# B&R Automation Studio project RS15_RX_30005_r00
Automation Studio 3.0.80.31 SP01

## Configuration Config1

### Acp10map.ncm - PLC1/Motion/Acp10map.ncm
```
NcMapping (NcSwId=acp10)
  NcObject Axis3 (ModuleAddress=SL1.SS1.IF2.ST3, InterfaceType=Powerlink, Type=ncAXIS, Channel=1, InitParameter=A3_Init, AcoposParameter=A3_Par, Disabled=FALSE, ModuleDisabled=FALSE)
  NcObject SL1.SS1.IF2.ST3.VAxis1 (ModuleAddress=SL1.SS1.IF2.ST3, InterfaceType=Powerlink, Type=ncV_AXIS, Channel=1, Disabled=TRUE, ModuleDisabled=FALSE)
  NcObject Axis4 (ModuleAddress=SL1.SS1.IF2.ST3, InterfaceType=Powerlink, Type=ncAXIS, Channel=2, InitParameter=A4_Init, AcoposParameter=A4_Par, Disabled=FALSE, ModuleDisabled=FALSE)
  NcObject SL1.SS1.IF2.ST3.VAxis2 (ModuleAddress=SL1.SS1.IF2.ST3, InterfaceType=Powerlink, Type=ncV_AXIS, Channel=2, Disabled=TRUE, ModuleDisabled=FALSE)
  NcObject Axis5 (ModuleAddress=SL1.SS1.IF2.ST5, InterfaceType=Powerlink, Type=ncAXIS, Channel=1, InitParameter=A5_Init, AcoposParameter=A5_Par, Disabled=FALSE, ModuleDisabled=FALSE)
  NcObject Axis9 (ModuleAddress=SL1.SS1.IF2.ST5, InterfaceType=Powerlink, Type=ncV_AXIS, Channel=1, InitParameter=A9_Init, AcoposParameter=A9_Par, Disabled=FALSE, ModuleDisabled=FALSE)
  NcObject Axis6 (ModuleAddress=SL1.SS1.IF2.ST5, InterfaceType=Powerlink, Type=ncAXIS, Channel=2, InitParameter=A6_Init, AcoposParameter=A6_Par, Disabled=FALSE, ModuleDisabled=FALSE)
  NcObject SL1.SS1.IF2.ST5.VAxis2 (ModuleAddress=SL1.SS1.IF2.ST5, InterfaceType=Powerlink, Type=ncV_AXIS, Channel=2, Disabled=TRUE, ModuleDisabled=FALSE)
  NcObject Axis1 (ModuleAddress=SL1.SS1.IF2.ST1, InterfaceType=Powerlink, Type=ncAXIS, Channel=1, InitParameter=A1_Init, AcoposParameter=A1_Par, Disabled=FALSE, ModuleDisabled=FALSE)
  NcObject SL1.SS1.IF2.ST1.VAxis1 (ModuleAddress=SL1.SS1.IF2.ST1, InterfaceType=Powerlink, Type=ncV_AXIS, Channel=1, Disabled=FALSE, ModuleDisabled=FALSE)
  NcObject SL1.SS1.IF2.ST1.Axis2 (ModuleAddress=SL1.SS1.IF2.ST1, InterfaceType=Powerlink, Type=ncAXIS, Channel=2, Disabled=FALSE, ModuleDisabled=FALSE)
  NcObject Axis11 (ModuleAddress=SL1.SS1.IF2.ST1, InterfaceType=Powerlink, Type=ncV_AXIS, Channel=2, InitParameter=A11_Init, AcoposParameter=A11_Par, Disabled=FALSE, ModuleDisabled=FALSE)
  NcObject SL1.SS1.IF2.ST2.Axis2 (ModuleAddress=SL1.SS1.IF2.ST2, InterfaceType=Powerlink, Type=ncAXIS, Channel=2, Disabled=FALSE, ModuleDisabled=FALSE)
  NcObject SL1.SS1.IF2.ST2.VAxis2 (ModuleAddress=SL1.SS1.IF2.ST2, InterfaceType=Powerlink, Type=ncV_AXIS, Channel=2, Disabled=TRUE, ModuleDisabled=FALSE)
  NcObject Axis2 (ModuleAddress=SL1.SS1.IF2.ST2, InterfaceType=Powerlink, Type=ncAXIS, Channel=1, InitParameter=A2_Init, AcoposParameter=A2_Par, Disabled=FALSE, ModuleDisabled=FALSE)
  NcObject Axis0 (ModuleAddress=SL1.SS1.IF2.ST10, InterfaceType=Powerlink, Type=ncAXIS, Channel=1, AcoposSimulation=Off, InitParameter=A0_Init, AcoposParameter=A0_Par, Disabled=FALSE, ModuleDisabled=FALSE)
  NcObject SL1.SS1.IF2.ST10.VAxis1 (ModuleAddress=SL1.SS1.IF2.ST10, InterfaceType=Powerlink, Type=ncV_AXIS, Channel=1, Disabled=TRUE, ModuleDisabled=FALSE)
  NcObject SL1.SS1.IF2.ST10.Axis2 (ModuleAddress=SL1.SS1.IF2.ST10, InterfaceType=Powerlink, Type=ncAXIS, Channel=2, AcoposSimulation=Off, Disabled=TRUE, ModuleDisabled=FALSE)
  NcObject SL1.SS1.IF2.ST10.VAxis2 (ModuleAddress=SL1.SS1.IF2.ST10, InterfaceType=Powerlink, Type=ncV_AXIS, Channel=2, Disabled=TRUE, ModuleDisabled=FALSE)
  NcObject SL1.SS1.IF2.ST2.VAxis1 (ModuleAddress=SL1.SS1.IF2.ST2, InterfaceType=Powerlink, Type=ncV_AXIS, Channel=1, Disabled=TRUE, ModuleDisabled=FALSE)
  NcObject Axis7 (ModuleAddress=SL1.SS1.IF2.ST7, InterfaceType=Powerlink, Type=ncAXIS, Channel=1, InitParameter=A7_Init, AcoposParameter=A7_Par, Disabled=FALSE, ModuleDisabled=FALSE)
  NcObject SL1.SS1.IF2.ST7.VAxis1 (ModuleAddress=SL1.SS1.IF2.ST7, InterfaceType=Powerlink, Type=ncV_AXIS, Channel=1, Disabled=TRUE, ModuleDisabled=FALSE)
  NcObject SL1.SS1.IF2.ST7.Axis2 (ModuleAddress=SL1.SS1.IF2.ST7, InterfaceType=Powerlink, Type=ncAXIS, Channel=2, Disabled=FALSE, ModuleDisabled=FALSE)
  NcObject SL1.SS1.IF2.ST7.VAxis2 (ModuleAddress=SL1.SS1.IF2.ST7, InterfaceType=Powerlink, Type=ncV_AXIS, Channel=2, Disabled=TRUE, ModuleDisabled=FALSE)
```

## Configuration Simul_AR000

### Task classes (Cpu.sw)
```
Cyclic#1:
  A9_Basic <- BagMachine_Section.MasterAxis.A9_Init.A9_Basic.prg
  A9_Control <- BagMachine_Section.MasterAxis.A9_Init.A9_Control.prg
  A15_Basic <- BagMachine_Section.HotMicroPerf.Axis15.A15_Basic.prg
  A15_Automa <- BagMachine_Section.HotMicroPerf.Axis15.A15_Automat.prg
Cyclic#4:
  A15_Contro <- BagMachine_Section.HotMicroPerf.Axis15.A15_Control.prg
  A15_Motion <- BagMachine_Section.HotMicroPerf.Axis15.A15_MotionCycle.prg
  HMPerf_Gen <- BagMachine_Section.HotMicroPerf.HMPerf_Gen.prg
  Test_Simul <- BagMachine_Section.BagBundler.Test_Simul.prg
DataObjects: arsdmsvp, arsdmsvg, arsdmhtm, Acp10sys
NcDataObjects: A9_Par <- BagMachine_Section.MasterAxis.A9_Init.A9_Par.dob, A15_Init <- BagMachine_Section.HotMicroPerf.Axis15.A15_Init.dob, A15_Par <- BagMachine_Section.HotMicroPerf.Axis15.A15_Par.dob, A9_Init <- BagMachine_Section.MasterAxis.A9_Init.A9_Init.dob, A1_Par, A1_Init
Binaries: arsdm, webserv, Acp10map, ashwd, sysconf, arconfig, iomap, asfw, Acp10cfg, vccnum, vcnet, HMI_10, HMI_1003, vcpdvnc, vcbclass, vcgclass, vccbtn, vcpfar00, vcshared, vccline, vccdt, vcalarm, vccddbox, vcfntttf, arialbd, vctcal, vccovl, vcdsloc, visvc, vccbmp, arial, vcpdsw, vcdsint, vcfile, vccshape, HMI_1001, vcmgr, vcresman, vccstr, visapi, vcchspot, vccpopup, vcrt, HMI_1002, arialbi, vcctext, vcclbox, vccalarm
Libraries: Brsystem, NcGlobal, HGWeber, astime, runtime, powerlnk, Acp10sdc, Acp10man, Acp10par, fileio, sys_lib, asmem, standard, convert, dataobj, astcp, Acp10_MC
```

## Logical view

Binary libraries used (declarations not repeated): Acp10_MC 3.18.2, Acp10man 3.18.2, Acp10par 3.18.2, Acp10sdc 3.18.2, AsMath, AsMem, asstring, astime, Brsystem, Convert, LoopConR 2.80.0, powerlnk, sys_lib

### Global.var
```iecst
(********************************************************************
 * COPYRIGHT --
 ********************************************************************
 * File: Global.var
 * Author: pkiel
 * Created: September 02, 2009
 ********************************************************************
 * Global variables of project NewAxisControl
 ********************************************************************)
VAR
	gA : ARRAY[0..15] OF AxisBasic;
END_VAR
VAR RETAIN
	gA1_FirstHomed : BOOL;
	gA11_FirstHomed : BOOL;
END_VAR
VAR
	gA1Ref_Horn : BOOL;
	gA1Ref_PB : BOOL;
END_VAR
VAR RETAIN
	gA2_FirstHomed : BOOL;
	gA3_FirstHomed : BOOL;
END_VAR
VAR
	gA3Ref_Horn : BOOL;
	gA3Ref_PB : BOOL;
END_VAR
VAR RETAIN
	gA4_FirstHomed : BOOL;
END_VAR
VAR
	gA4Ref_PB : BOOL;
	gA4Ref_Horn : BOOL;
END_VAR
VAR RETAIN
	gA5_FirstHomed : BOOL;
END_VAR
VAR
	gA5_GearValue : REAL;
	gA5Ref_Horn : BOOL;
	gA5Ref_PB : BOOL;
END_VAR
VAR RETAIN
	gA6_FirstHomed : BOOL;
END_VAR
VAR
	gA6_GearValue : REAL;
	gA6Ref_Horn : BOOL;
	gA6Ref_PB : BOOL;
	gA8_GearValue : REAL;
	gA8Ref_Horn : BOOL;
	gA8Ref_PB : BOOL;
END_VAR
VAR RETAIN
	gA7_FirstHomed : BOOL;
END_VAR
VAR
	gA7Ref_Horn : BOOL;
	gA7Ref_PB : BOOL;
	gA13Ref_Horn : BOOL;
	gA13Ref_PB : BOOL;
	gA13_RefDone : BOOL;
	gA12Ref_Horn : BOOL;
	gA12Ref_PB : BOOL;
	gA12_RefDone : BOOL;
END_VAR
VAR RETAIN
	gA13_FirstHomed : BOOL;
	gA12_FirstHomed : BOOL;
	gA8_FirstHomed : BOOL;
	gA9_FirstHomed : BOOL;
END_VAR
VAR
	gA9Ref_Horn : BOOL;
	gA9Ref_PB : BOOL;
END_VAR
VAR RETAIN
	gA10_FirstHomed : BOOL;
END_VAR
VAR
	gA10Ref_Horn : BOOL;
	gA10Ref_PB : BOOL;
END_VAR
VAR RETAIN
	gA14_FirstHomed : BOOL;
END_VAR
VAR
	gA14_RefDone : BOOL;
END_VAR
VAR RETAIN
	gA16_FirstHomed : BOOL;
END_VAR
VAR
	gA15_RefDone : BOOL;
	gA15Ref_Horn : BOOL;
	gA15Ref_PB : BOOL;
	gA2_RefDone : BOOL;
	gA2Ref_Horn : BOOL;
	gA2Ref_PB : BOOL;
END_VAR
VAR RETAIN
	gA15_FirstHomed : BOOL;
END_VAR
VAR
	gA16_RefDone : BOOL;
	gActualMachineSpeed_BPM : REAL;
	gActualMachineSpeed_FPM : REAL;
	gAlarmReset : BOOL;
	gAlarmsOK : BOOL;
	gBagMachine_AlarmsOK : BOOL;
	gBagMachine_EstopAlarmsOK : BOOL;
	gBagMachine_GuardAlarmsOK : BOOL;
	gBagMachine_IOAlarmsOK : BOOL;
  gBagMachine_JamAlarmsOK : BOOL;
  gBagMachine_MotorAlarmsOK : BOOL;
  g_bBagMachine_GenAlarmsOK : BOOL;
	g_bBagMachine_EndReelAlarmsOK : BOOL;
	g_bBagMachine_DryerAlarmsOK : BOOL;
  g_bBagMachine_CamProfCalcOK : BOOL;
END_VAR
VAR CONSTANT
	gBlack : UINT := 0;
	gBlue : UINT := 1;
END_VAR
VAR
	gCurrentScreen : UINT;
	gDriveSupply_Ready : BOOL;
END_VAR
VAR RETAIN
	gEndPosData : ARRAY[0..15] OF MC_ENDLESS_POSITION;
END_VAR
VAR
	gEStopAlarmsOK : BOOL;
	gFastStop_OK : BOOL;
	gGeneralFaults_OK : BOOL;
  gGluerAlarmsOK : BOOL;
  g_bGenAlarmsOK : BOOL;
END_VAR
VAR CONSTANT
	gGray : UINT := 59;
	gGray1 : UINT := 250;
	gGreen : UINT := 10;
END_VAR
VAR
	gGuardAlarmsOK : BOOL;
	gGuardsOK : BOOL;
END_VAR
VAR RETAIN
	gHMI_CmdSpeed : REAL;
END_VAR
VAR
	gHMI_GoToHoldTearDrum_PB : BOOL := FALSE;
	gHMI_GoToAlarm_PB : BOOL := FALSE;
	gHMI_GoToMain_PB : BOOL := FALSE;
	gHMI_GoToMaint_PB : BOOL := FALSE;
	gHMI_GoToSetup_PB : BOOL := FALSE;
	gHMI_GoToStatus_PB : BOOL := FALSE;
	gHMI_Jog_PB : BOOL := FALSE;
	gHMI_PasswordLevel : INT;
	gHMI_Reset_PB : BOOL := FALSE;
	gHMI_Run_PB : BOOL := FALSE;
	gHMI_Stop_PB : BOOL := FALSE;
	gI_E1_Spare1 : BOOL := FALSE;
	gI_E1_Spare2 : BOOL := FALSE;
	gI_E1_Spare3 : BOOL := FALSE;
	gI_E1_Spare4 : BOOL := FALSE;
	gAI_E1_Spare1 : INT := 0;
	gAI_E1_Spare2 : INT := 0;
	gI_L3_Spare1 : BOOL := FALSE;
	gI_L3_Spare2 : BOOL := FALSE;
	gI_L3_Spare3 : BOOL := FALSE;
	gI_L3_Spare4 : BOOL := FALSE;
	gAI_L3_Spare1 : INT := 0;
	gAI_L3_Spare2 : INT := 0;
	gI_230Vac_OK : BOOL := FALSE;
	gI_AirPressureOK : BOOL := FALSE;
	gI_EstopPB_1 : BOOL := FALSE; (*+R4*)
	gI_EstopPB_2 : BOOL := FALSE; (*+R3*)
	gI_EstopPB_3 : BOOL := FALSE; (*+R1*)
	gI_EstopPB_4 : BOOL := FALSE; (*+R2*)
	gI_EstopPB_5 : BOOL := FALSE; (*+R1A*)
	gI_EstopPB_Unwind : BOOL := FALSE;
	gI_FasterPB_1 : BOOL := FALSE;
	gI_FstopPB_1 : BOOL := FALSE;
	gI_GSW_Door1 : BOOL := FALSE;
	gI_GSW_Door2 : BOOL := FALSE;
	gI_GSW_Drum : BOOL := FALSE;
	gI_GSW_PerfDoors : BOOL := FALSE;
	gI_GSW_PerfDoor2 : BOOL := FALSE;
	gI_GSW_RSEntry : BOOL := FALSE;
	gI_GSW_SlittingDoor : BOOL := FALSE;
	gI_GSW_Tearing : BOOL := FALSE;
	gI_JamPE_RS : BOOL := FALSE;
	gI_JogPB_1 : BOOL := FALSE;
	gI_MP_DrumFan : BOOL := FALSE;
	gI_MP_GlueSlowRotation : BOOL := FALSE;
	gI_MP_PerfFan : BOOL := FALSE;
	gI_MP_Vacuum : BOOL := FALSE;
	gI_PB_MachineStart : BOOL := FALSE;
	gI_ResetPB_1 : BOOL := FALSE;
	gCmd_ResetPBGen : BOOL := FALSE; (*General reset all failures*)
	gI_SafetyRelay_EStopOK : BOOL := FALSE;
	gI_SafetyRelay_GuardOK : BOOL := FALSE;
	gI_SlowerPB_1 : BOOL := FALSE;
	gI_SlowerPB_2 : BOOL := FALSE;
	gI_SS_DrumNeg : BOOL := FALSE;
	gI_SS_DrumPos : BOOL := FALSE;
	gI_SS_ExitTableFaster : BOOL := FALSE;
	gI_SS_ExitTableSlower : BOOL := FALSE;
	gI_SS_GluePanUpDown : BOOL := FALSE;
	gI_SS_HoldingNeg : BOOL := FALSE;
	gI_SS_HoldingPos : BOOL := FALSE;
	gI_SS_MainPowerOff : BOOL;
	gI_SS_MainPowerOn : BOOL := FALSE;
	gI_SS_PerfNeg : BOOL := FALSE;
	gI_SS_PerfPos : BOOL := FALSE;
	gI_SS_SeamGlueOnOff : BOOL := FALSE;
	gI_PrintOn_PB : BOOL := FALSE;
	gI_PrintOff_PB : BOOL := FALSE;
	gI_SS_TearingNeg : BOOL := FALSE;
	gI_SS_TearingPos : BOOL := FALSE;
	gI_SS_WebEntryNipOff_1 : BOOL := FALSE;
	gI_SS_WebEntryNipOff_2 : BOOL := FALSE;
	gI_SS_WebEntryNipOn_1 : BOOL := FALSE;
	gI_SS_WebEntryNipOn_2 : BOOL := FALSE;
	gI_SS_WebExitNip : BOOL := FALSE;
	gI_StopPB_1 : BOOL := FALSE;
	gI_StopPB_2 : BOOL := FALSE;
	gI_StopPB_3 : BOOL := FALSE; (*Stop PB on +R2 panel*)
	gI_JogPB_2 : BOOL := FALSE; (*Footswitch Job*)
	gI_JogPB_3 : BOOL := FALSE; (*Flexo press Job*)
	gI_WebBreakPE_1 : BOOL := FALSE;
	gI_WebBreakPE_2 : BOOL := FALSE;
	gI_EstopPB_FlexoPress : BOOL := FALSE;
	gI_UNW_EndReelPolyPE : BOOL := FALSE;
	gI_UNW_EndReelPapPE : BOOL := FALSE;
	gI_SS_UNW_ForkUp : BOOL := FALSE;
	gI_SS_UNW_ForkDown : BOOL := FALSE;
	gI_SS_UNW_Brake : BOOL := FALSE;
	gI_MP_UNW_HydroPump : BOOL := FALSE;
	gI_SS_UNW_HotGlue : BOOL := FALSE;
	gI_SS_FP_NipRol : BOOL := FALSE;
	gI_MP_FP_MotorFan : BOOL := FALSE;
	gI_FP_PrintOn_PB : BOOL := FALSE;
	gI_FP_PrintOff_PB : BOOL := FALSE;
	gI_MP_FP_SlowRot5 : BOOL := FALSE;
	gI_MP_FP_SlowRot6 : BOOL := FALSE;
	gI_GSW_FP_Doors : BOOL := FALSE;
	gI_GSW_FP_Gates : BOOL := FALSE;
	gI_MP_FP_SlowRot1 : BOOL := FALSE;
	gI_MP_FP_SlowRot3 : BOOL := FALSE;
	gI_MP_FP_SlowRot2 : BOOL := FALSE;
	gI_MP_FP_SlowRot4 : BOOL := FALSE;
	gI_HMP_BrushReturnPE : BOOL := FALSE;
	gI_HMP_ProtecDownPE : BOOL := FALSE;
	gI_SS_HMPerfNeg : BOOL := FALSE;
	gI_SS_HMPerfPos : BOOL := FALSE;
	gI_HMP_On_PB : BOOL := FALSE;
	gI_HMP_Off_PB : BOOL := FALSE;
	gI_HMP_EStopPB : BOOL := FALSE;
	gI_SS_HMP_Heating : BOOL := FALSE;
	gI_GSW_HMPerf : BOOL := FALSE;
	gI_SS_HMP_ManuProtecDown : BOOL := FALSE;
	gI_HMP_ManuBrushForward_PB : BOOL := FALSE;
	gI_HMP_WebBreakPE : BOOL := FALSE;
	gI_HMP_JogPB : BOOL := FALSE;
	gI_L15_Spare1 : BOOL := FALSE;
	gI_L15_Spare2 : BOOL := FALSE;
	gI_L15_Spare3 : BOOL := FALSE;
	gI_L15_Spare4 : BOOL := FALSE;
	gI_SS_3W_GlueOn : BOOL := FALSE;
	gI_SS_3W_Glue2 : BOOL := FALSE;
	gI_MP_HP_WasteSuction : BOOL := FALSE;
	gI_3W_EndReelPolyPE : BOOL := FALSE;
	gI_MP_3W_Fan : BOOL := FALSE;
	gI_3W_EStopPB : BOOL := FALSE;
	gI_GSW_3W : BOOL := FALSE;
	gI_SS_3W_FanOnOff : BOOL := FALSE;
	gI_DRY_Thermostat : BOOL := FALSE;
	gI_MP_DRY_Blower : BOOL := FALSE;
	gI_MP_DRY_Heater : BOOL := FALSE;
	gI_E1_Spare6  : BOOL := FALSE;
  gI_E1_Spare5  : BOOL := FALSE;
  gI_E1_Spare7  : BOOL := FALSE;
  gI_E1_Spare8  : BOOL := FALSE;
  gI_E1_Spare9  : BOOL := FALSE;
  gI_E1_Spare10 : BOOL := FALSE;
	gI_L3_Spare5 : BOOL := FALSE;
	gI_L3_Spare6 : BOOL := FALSE;
	gI_L3_Spare7 : BOOL := FALSE;
	gI_GSW_CMPerfDoor : BOOL := FALSE;
	gI_GSW_CMPerfGates : BOOL := FALSE;
	gI_MP_EB_WasteSuction : BOOL := FALSE;
	gI_SS_EnvBagNeg : BOOL := FALSE;
	gI_SS_EnvBagPos : BOOL := FALSE;
	gI_SS_TearEBNeg : BOOL := FALSE;
	gI_SS_TearEBPos : BOOL := FALSE;
	gAI_DRY_Pt100_Temp : INT;
END_VAR
VAR RETAIN
	gMachineTime : HourMeter;
END_VAR
VAR
	gMaintDropdown : UINT;
	gMaintScreenChange : BOOL;
	gManualMode_On : BOOL;
	gMotorAlarmsOK : BOOL;
	gNever : BOOL;
	gNever1 : BOOL; (*D.M. 05/08/2011 Inibit function BrownPaper_14542*)
END_VAR
VAR RETAIN
	gPassword : PasswordLevel;
END_VAR
VAR
	gPerf_On : BOOL;
	gPerf_ParkRequest : BOOL;
END_VAR
VAR RETAIN
	gPerf_ParkRequired : BOOL;
END_VAR
VAR
	gPerfSelect_Large : BOOL;
	gPowerUp_Complete : BOOL;
END_VAR
VAR CONSTANT
	gPurple : UINT := 62;
END_VAR
VAR
	gQ_E1_Spare1 : BOOL := FALSE;
	gQ_E1_Spare2 : BOOL := FALSE;
  gQ_E1_Spare3 : BOOL := FALSE;
  gQ_E1_Spare4 : BOOL := FALSE;
  gQ_E1_Spare5 : BOOL := FALSE;
  gQ_E1_Spare6 : BOOL := FALSE;
	gAQ_E1_Spare1 : INT := 0;
	gAQ_E1_Spare2 : INT := 0;
	gQ_L3_Spare1 : BOOL := FALSE;
	gQ_L3_Spare2 : BOOL := FALSE;
  gQ_L3_Spare3 : BOOL := FALSE;
  gQ_L3_Spare4 : BOOL := FALSE;
  gQ_L3_Spare5 : BOOL := FALSE;
  gQ_L3_Spare6 : BOOL := FALSE;
	gAQ_L3_Spare1 : INT := 0;
	gAQ_L3_Spare2 : INT := 0;
	gQ_CMD_ColdGluePressure : INT := 0;
	gQ_CMD_EjectionTableMotor : INT := 0;
	gQ_CMD_HotGluePressure : INT := 0;
	gQ_CMD_RS_GluePressure : INT := 0;
	gQ_CMD_UNW_GluePressure : INT := 0;
	gQ_CMD_3W_GluePressure : INT := 0;
	gQ_CMD_OtherRS_GluePressure : INT := 0;
	gQ_CMD_RS_ExitTableSpeed : INT := 0;
	gQ_CON_GlueSlowRotation : BOOL := FALSE;
	gQ_CON_Vacuum : BOOL := FALSE;
	gQ_CR_ColdGlue : BOOL := FALSE;
	gQ_CR_ColdGlueSelect : BOOL := FALSE;
	gQ_CR_EstopReset : BOOL := FALSE;
	gQ_CR_GuardBypass : BOOL := FALSE;
	gQ_CR_HotGlue : BOOL := FALSE;
	gQ_CR_HotGlueSelect : BOOL := FALSE;
	gQ_CR_MainPowerOn : BOOL := FALSE;
	gQ_CR_UnwinRegEnable : BOOL := FALSE; (*Enable regulation on the unwinder*)
	gQ_CR_WarningHorn : BOOL := FALSE;
	gQ_CR_WatchDog : BOOL := FALSE;
	gQ_PL_GenFailure : BOOL := FALSE;
	gQ_PL_MainPower : BOOL := FALSE;
	gQ_SOL_BagCount : BOOL := FALSE;
	gQ_SOL_GluePan : BOOL := FALSE;
	gQ_SOL_WebEntryNip : BOOL := FALSE;
	gQ_SOL_WebExitNip : BOOL := FALSE;
	gQ_CR_UNW_HydroPump : BOOL := FALSE;
	gQ_CR_HotColdRSGlueSelect : BOOL := FALSE;
	gQ_CR_HotColdOtherRSGlueSelect : BOOL := FALSE;
	gQ_CR_UNW_Brake : BOOL := FALSE; (*MEROBEL device input B*)
	gQ_CR_FP_NipRol : BOOL := FALSE;
	gQ_CR_FP_Print : BOOL := FALSE;
	gQ_CR_UNW_PIDRegul : BOOL := FALSE; (*MEROBEL device input A*)
	gQ_CR_UNW_ForkUp : BOOL := FALSE;
	gQ_CR_UNW_ForkDown : BOOL := FALSE;
	gQ_CR_RS_Glue : BOOL := FALSE;
	gQ_CR_UNW_Glue : BOOL := FALSE;
	gQ_SOL_HMP_BrushForward : BOOL := FALSE;
	gQ_SOL_HMP_ProtecDown : BOOL := FALSE;
	gQ_HMP_LightOn : BOOL := FALSE;
	gQ_HMP_Heater : BOOL := FALSE;
	gQ_CR_3W_GlueOn : BOOL := FALSE;
	gQ_CR_3W_Glue2 : BOOL := FALSE;
	gQ_CR_3W_Fan : BOOL := FALSE;
	gQ_CR_HP_WasteSuction : BOOL := FALSE;
	gQ_CR_DRY_Blower : BOOL := FALSE;
	gQ_CR_DRY_HeatRegul : BOOL := FALSE;
	gQ_CR_DRY_HeatContinu : BOOL := FALSE;
	gQ_CR_EB_WasteSuction : BOOL := FALSE;
	gQ_CR_UNW_Lock : BOOL := FALSE;
END_VAR
VAR RETAIN
	gRecipeActive : Recipe := (rEnvB_PerfSize_in:=18.897); (*Default Envelope Bag Perf Size = 480mm Customer Pyrollpack_14661*)
	gRecipeBase : ARRAY[0..50] OF Recipe;
END_VAR
VAR
	gRecipeChange : BOOL;
	gRecipeCntl : RECIPE_CNTL_typ;
END_VAR
VAR CONSTANT
	gRed : UINT := 51;
END_VAR
VAR RETAIN
	gReg : ARRAY[0..15] OF Registration;
END_VAR
VAR
	gInchMetric_Ind : UINT; (*=1:Inch, =2:Metric*)
	gIOAlarmsOK : BOOL;
	gJamAlarmsOK : BOOL;
	gWebBreakAlarmsOK : BOOL;
	gJog_Horn : BOOL;
	gJog_ToZeroFiltered : BOOL;
	gRun_Stop : BOOL;
	gJog_Stop : BOOL;
	gJog_ToZeroSpeed : BOOL;
	gMachine_Jog : BOOL;
	gMachine_Run : BOOL;
	gMachineMaxSpeedLimit : REAL;
	gMachineMinSpeedLimit : REAL;
	gRepeatChange : BOOL;
	gRun_Horn : BOOL;
	gRun_ToZeroSpeed : BOOL;
	gScreenControl : UINT;
	gServoAxesOK : BOOL;
	gSetupMode_On : BOOL;
	gSetupPermissive : BOOL;
END_VAR
VAR RETAIN
	gSP_A : ARRAY[0..15] OF AxisSP := [(HomeOffset:=0.0,PhaseOffset:=0.0,Diameter:=0.0,ParkPosition:=0.0,MatchedSpeed:=0.0,AbsoluteOffset:=0.0,rZoneBefPerf_in:=0.0,rZoneAftPerf_in:=0.0),(HomeOffset:=120.0,ParkPosition:=120.0,MatchedSpeed:=60.0),(HomeOffset:=0.0,PhaseOffset:=0.0,Diameter:=0.0,ParkPosition:=0.0,MatchedSpeed:=0.0,AbsoluteOffset:=0.0,rZoneBefPerf_in:=0.0,rZoneAftPerf_in:=0.0),2((HomeOffset:=20.0)),2((HomeOffset:=0.0,PhaseOffset:=0.0,Diameter:=0.0,ParkPosition:=0.0,MatchedSpeed:=0.0,AbsoluteOffset:=0.0,rZoneBefPerf_in:=0.0,rZoneAftPerf_in:=0.0)),(HomeOffset:=20.0),(HomeOffset:=20.0,PhaseOffset:=0.0,Diameter:=0.0,ParkPosition:=0.0,MatchedSpeed:=0.0,AbsoluteOffset:=0.0,rZoneBefPerf_in:=0.0,rZoneAftPerf_in:=0.0),4((HomeOffset:=0.0,PhaseOffset:=0.0,Diameter:=0.0,ParkPosition:=0.0,MatchedSpeed:=0.0,AbsoluteOffset:=0.0,rZoneBefPerf_in:=0.0,rZoneAftPerf_in:=0.0)),(HomeOffset:=20.0,PhaseOffset:=0.0,Diameter:=0.0,ParkPosition:=0.0,MatchedSpeed:=0.0,AbsoluteOffset:=0.0,rZoneBefPerf_in:=0.0,rZoneAftPerf_in:=0.0),2((HomeOffset:=0.0,PhaseOffset:=0.0,Diameter:=0.0,ParkPosition:=0.0,MatchedSpeed:=0.0,AbsoluteOffset:=0.0,rZoneBefPerf_in:=0.0,rZoneAftPerf_in:=0.0))];
	gSP_EnvBPerf : AxisSP; (*Envelope Bag Perf*)
	gSP_StandPerf : AxisSP; (*Standard Perf*)
	gSP_CmdSpeed : REAL;
	gSP_ColdGlue : Glue;
	gSP_RSGlue : Glue;
	gSP_OtherRSGlue : Glue;
	gSP_GlueTrayAutoSpeed : REAL;
	gSP_HotGlue : Glue;
	gSP_PerfCylSelect : BOOL; (*Perf Size selection =0:Small; =1:Large*)
	gSP_PerfKnifeCount : REAL;
	gSP_TubeSelect : BOOL;
END_VAR
VAR
	gStopPosition : REAL;
	gStopStringOK : BOOL;
	gTubeSelect_2 : BOOL;
	gUnwindLowRoll_Stop : BOOL;
	gBagMachine_WebBreakOK : BOOL;
	gWebBreakBypass_On : BOOL;
	g_bEndReelPapBypass_On : BOOL;
	g_bEndReelPolyBypass_On : BOOL;
	g_rActualSizePerf_in : REAL; (*Actual perimeter of the Perf, in inch*)
	g_bPerfInMatchedSpeed : BOOL;
	g_bMainPower_On : BOOL;
	g_bMainPower_OnDelay : BOOL;
  g_bCamPerfCalc_Error : BOOL;
  g_bCamPerfCalcReset : BOOL;
  g_uiCalcCamPerfErrorID : UINT;
  g_bMachineRun : BOOL;
  g_bCameProf_OK : BOOL;
  g_uiIndexCamProfPerf : UINT;
  g_uiGetPosCamProfErrorID_1 : UINT;
  g_uiGetPosCamProfErrorID_2 : UINT;
  g_uiGetPosCamProfErrorID_3 : UINT;
  g_uiHomCamProfErrorID : UINT;
  g_bGetMaPosCamProfError_1 : BOOL;
  g_bGetMaPosCamProfError_2 : BOOL;
  g_bHomeCamProfError : BOOL;
  g_uiGetPosCamProfErrorID : UINT;
  g_bGetMaPosCamProfError : BOOL;
  g_bGetSlPosCamProfError : BOOL;
  g_rPosParkMasterCam : REAL ;
	g_bIndSynchroHTD_OK : BOOL; (*Indicator synchro Holding, Tearing and Drum axis is completed*)
	g_iMachType : INT; (*Machine type : =1:RS26, =2:RS15, =3:RS25*)
	g_iFlexoType : INT; (*Flexo type : =0:Metric, =1:8DP, =2:10DP, =3:1/4"*)
	g_bIndEStop : BOOL; (*EStop active*)
	g_bIndEStopStandstill : BOOL; (*EStop when machine at standstill*)
	g_bIndStopFault : BOOL; (*Machine stopping on fault condition*)
  g_bUnwindInMach : BOOL;
  g_bUnwindEndRelPapInMach : BOOL;
  g_bUnwindEndRelPolyInMach : BOOL;
	g_bFP_IndSpeedLimit : BOOL; (*Speed limited because max speed Flexo Press reached*)
	g_rNumbPliers : REAL; (*Number of pliers on the Drum, 4 or 2*)
	g_bNumPliersChange : BOOL;
	g_bNumPliersChange2to4 : ARRAY[1..3] OF BOOL; (*Change number of pliers on the Drum, from 2 to 4*)
	g_bNumPliersChange4to2 : ARRAY[1..3] OF BOOL; (*Change number of pliers on the Drum, from 4 to 2*)
	g_bChangeModTearingReq : BOOL; (*Change modulus on tearing axis request*)
	g_bChangeModTearEBReq : BOOL; (*Change modulus on Tearing Envelope Bag axis request*)
	g_bChangeModDrumReq : BOOL; (*Change modulus on tearing axis request*)
	g_bRedefPosdTearingReq : BOOL; (*Redefinition of the position on Tearing axis request*)
	g_bRedefPosDrumReq : BOOL; (*Redefinition of the position on Drum axis request*)
	g_bSynchroAxisOK : BOOL; (*All axis are synchro*)
	g_bSynchroAxisInProgress : BOOL; (*Synchro axis in progress*)
	g_rMaxBagSize_Inch : REAL;
	g_rMinBagSize_Inch : REAL;
	g_bSplashDone : BOOL;
	g_b3WebUnitInMach : BOOL;
	g_bFP_NipRolAutoOff : BOOL;
	g_bFP_GuardFault : BOOL;
	g_bLockSP_OffsetPrintRol : BOOL;
	g_bFP_SP_Offset : BOOL; (*Change Offset of the Flexo with set point motion*)
	g_rPrintRolCalcPos_deg : REAL; (*Calculated position of the printing rolle, in °*)
	g_rPrintRolCalcPos_in : REAL; (*Calculated position of the printing rolle, in inch*)
	g_HMI_Cmd_ManuTimSetPlus : BOOL;
	g_bCondManuTimSet : BOOL;
	g_bStartOffsetAuto : BOOL;
	g_rZGearRepFP : REAL := 40.0; (*Current tooth number of the gear on the Flexo Press*)
	g_bCmdShiftA : ARRAY[1..15] OF BOOL; (*Command shift Axe[n]*)
	g_iCountPerfShift : ARRAY[1..2] OF INT; (*Counter of Perf shifting in order to match with printing position*)
	g_iNumBagPerfTear : INT; (*Num bags between Perf en teraing > gr_rDistPerfTear_mm / BagSize example : 3800/200 = 19*)
	g_iArrayBagPerfTear : ARRAY[0..C_iMaxBagPerfTear] OF INT; (*Array of bags between Perf and tearing, +1 for positive shift and -1 for negative shift*)
	g_iArrayBagPerfTearNul : ARRAY[0..C_iMaxBagPerfTear] OF INT := [C_iMaxBagPerfTear(0)]; (*Array with all elements C_iMaxBagPerfTear =0*)
	gr_rIndEnvB2AxTear1 : BOOL := 0; (*Envelope Bag 2 Axes, indicator tearin on the first station (tube lenght > gr_rEnvBSizeTear2_1_mm), =0:NO; =1:YES *)
	g_bPerfShiftPos : BOOL;
	g_iPerfShiftPos : INT;
	g_bCycManTimeSetOn : BOOL; (*Indicator at least one manual timing setting is active*)
	g_bIndPhasDrumInact : BOOL := 0; (*Indicator phasing Drum inactive*)
	g_rZGearCMPerf : REAL; (*Current number of tooth on the gear which drive the Cold Micro Perf Tool*)
	g_rSizeCMPerf : REAL; (*Current number of tooth on the gear which drive the Cold Micro Perf Tool*)
	g_rSizeCMPerfRol_mm : REAL; (*Perimeter of the shaft which drive the Cold Micro Perf Tool, in mm*)
	g_iCMPerfType : INT; (*Cold Micro Perf type : =0:Metric, =1:8DP, =2:10DP, =3:1/4"*)
	g_stHMPerfCyc : CycHMPerf;
	g_bHMP_WebBreakBypass_On : BOOL;
	g_bHMP_CamOK : BOOL;
	g_bHMP_CamCalcReset : BOOL;
	g_bHMP_CamErrorGen : BOOL;
	g_bHMP_CamCalc_Error : BOOL;
	g_uiHMP_CalcCamErrorID : UINT;
	g_bHMP_CamDownl_Error : BOOL;
	g_uiHMP_DownlCamErrorID : UINT;
	g_bHMP_CmdPhasing : BOOL; (*Hot Micro Perf Phasing command to set the Offset when synchronizing*)
	g_bHMP_PhasInProgres : BOOL; (*Hot Micro Perf Phasing in progress to set the Offset when synchronizing*)
	g_rHMP_SP_Phasing : REAL; (*Hot Micro Perf Phasing Phasing Set Point to set the Offset when synchronizing, in Deg*)
	g_bDryerInMach : BOOL;
	g_bHeatDryInMach : BOOL;
	g_bSelDryerProd : BOOL;
	g_usiAI_DRY_Pt100_TempStatus : USINT;
	g_DRY_bTempSensorAlarm : BOOL;
	g_DRY_bHeaterAlarm : BOOL;
  g_DRY_bBlowerAlarm : BOOL;
  g_DRY_bActHeat : BOOL;
  g_DRY_bIndCooling : BOOL;
  g_DRY_bMemPowerOff : BOOL;
  g_DRY_bFlash : BOOL ;
	g_iPerfType : INT;
	g_bEnvBagSelectChang : BOOL;
	g_EnvB_bWasteSucMPAlarm : BOOL;
	g_EnvB_iHoldTearEnvBCase : INT;
END_VAR
VAR CONSTANT
	C_iRS26 : INT := 1;
	C_iRS15 : INT := 2;
	C_iRS25 : INT := 3;
	C_iM : INT := 0;
	C_i8DP : INT := 1;
	C_i10DP : INT := 2;
	C_i1_4P : INT := 3;
	gWhite : UINT := 15;
	gViolet_5 : UINT := 5;
	gYellow : UINT := 46;
	C_rMaxAna : REAL := 32767.0;
	C_iMaxBagPerfTear : INT := 39; (*Num max bags between > MaxDistPerfTear / MinBagSize = Around(4000/105) = 39*)
END_VAR
VAR RETAIN
	g_rBagSize1to2SPerf_in : REAL := 7.480; (*Bag Size for switching 1 --> 2 blades on the Perfo (1if >; 2 if <=) case Small Perfo, in in*)
	g_rBagSize1to2LPerf_in : REAL := 10.236; (*Bag Size for switching 1 --> 2 blades on the Perfo (1if >; 2 if <=) case Large Perfo, in mm*)
	g_rLinSpeedMin_ftmin : REAL := 32.808; (*Value of the Minimum Speed, in ft/min*)
END_VAR
VAR CONSTANT
	PI : REAL := 3.14159;
END_VAR
VAR
	g_rLinSpeedMin_bgmin        : REAL := 0.0; (*Value of the Minimum Speed, in bg/min*)
	g_rBagSize1to2SPerf_mm      : REAL := 190.0; (*Bag Size for switching 1 --> 2 blades on the Perfo (1if >; 2 if <=) case Small Perfo, in mm*)
	g_rBagSize1to2LPerf_mm      : REAL := 260.0; (*Bag Size for switching 1 --> 2 blades on the Perfo (1if >; 2 if <=) case Large Perfo, in mm*)
	g_rLinSpeedMin_mmin         : REAL := 10.0; (*Value of the Minimum Line Speed, in m/min*)
	g_rMaxSpeedMin_bpm          : REAL := 35.0; (*Value of the max bag/min at minimum speed, in bag/min*)
	g_rMaxSpeedSynchro_bpm      : REAL := 8.0; (*Value of the max bag/min when synchronising, in bag/min*)
	g_rMaxJogDecel_bpmm         : REAL := 1200.0; (*Value of the max Jog deceleration, in bag/min²*)
	g_rLinSpeedSP_AccRS26           : REAL := 600.0; (*Value of Line Speed SP accel, in m/min²*)
	g_rLinSpeedSP_DecRS26           : REAL := 600.0; (*Value of Line Speed SP decel, in m/min²*)
	g_rLinSpeedSP_JogDecRS26        : REAL := 2500.0; (*Value of Line Speed SP Jog decel, in m/min²*)
	g_rLinSpeedSP_EStopDecRS26      : REAL := 6000.0; (*Value of Line Speed SP EStop decel, in m/min²*)
	g_rLinSpeedSP_GuardFaultDecRS26 : REAL := 4500.0; (*Value of Line Speed SP Guard Fault decel, in m/min²*)
	g_rLinSpeedSP_WebBreakDecRS26   : REAL := 5200.0; (*Value of Line Speed SP EStop decel, in m/min²*)
	g_rLinSpeedSP_GenFaultDecRS26   : REAL := 3000.0; (*Value of Line Speed SP General Fault decel, in m/min²*)
  g_rLinSpeedSP_FStopDecRS26      : REAL := 1800.0; (*Value of Line Speed SP Fast Stop decel, in m/min²*)
  g_rLinSpeedSP_AccRS15           : REAL := 33.3; (*Value of Speed SP accel, in m/min/s => 0-->1000bag/min in 30s*)
  g_rLinSpeedSP_DecRS15           : REAL := 33.3; (*Value of Speed SP decel, in m/min/s => 0-->1000bag/min in 30s*)
  g_rLinSpeedSP_JogDecRS15        : REAL := 140.0; (*Value of SP Jog decel, in m/min/s => 1000-->0bag/min in 7s*)
  g_rLinSpeedSP_EStopDecRS15      : REAL := 333; (*Value of Speed SP EStop decel, in m/min/s => 1000-->0bag/min in 3s*)
  g_rLinSpeedSP_GuardFaultDecRS15 : REAL := 250.0; (*Value of Speed SP Guard Fault decel, in m/min/s => 1000-->0bag/min in 4s*)
  g_rLinSpeedSP_WebBreakDecRS15   : REAL := 250.0; (*Value of Speed SP EStop decel, in m/min/s => 1000-->0bag/min in 4s*)
  g_rLinSpeedSP_GenFaultDecRS15   : REAL := 167.0; (*Value of Speed SP General Fault decel, in m/min/s => 1000-->0bag/min in 6s*)
  g_rLinSpeedSP_FStopDecRS15      : REAL := 100.0; (*Value of Speed SP Fast Stop decel, in m/min/s => 1000-->0bag/min in 10s*)
  g_rSizeEntryPullRol_mm      : REAL := 400.0; (*Perimeter of the entry pull roll, in mm*)
	g_rSizeExitPullRol_mm       : REAL := 320.0; (*Perimeter of the exit pull roll, in mm*)
	g_rSizeLPerf_mm       : REAL := 400.0; (*Perimeter of the large Perf, in mm*)
	g_rSizeSPerf_mm       : REAL := 270.0; (*Perimeter of the small Perf, in mm*)
	g_rSizeDrum_mm        : REAL := 1680.0; (*Perimeter of the Drum, in mm*)
	g_rZGearRepFP_M       : REAL := 40.0; (*Tooth number of the gear on the Flexo Press in case Metric*)
	g_rZGearRepFP_8DP     : REAL := 40.0; (*Tooth number of the gear on the Flexo Press in case 8DP*)
	g_rZGearRepFP_10DP    : REAL := 50.0; (*Tooth number of the gear on the Flexo Press in case 10DP*)
	g_rZGearRepFP_1_4P    : REAL := 65.0; (*Tooth number of the gear on the Flexo Press in case 1/4"*)
	g_rZGearCMPerf_M      : REAL := 50.0; (*Tooth number of the gear on the shaft which drive the Cold Micro Perf Tool in case Metric*)
	g_rZGearCMPerf_8DP    : REAL := 50.0; (*Tooth number of the gear on the shaft which drive the Cold Micro Perf Tool in case 8DP*)
	g_rZGearCMPerf_10DP   : REAL := 63.0; (*Tooth number of the gear on the shaft which drive the Cold Micro Perf Tool in case 10DP*)
	g_rZGearCMPerf_1_4P   : REAL := 81.0; (*Tooth number of the gear on the shaft which drive the Cold Micro Perf Tool in case 1/4"*)
  g_rMaxBagSize_RS15_mm : REAL := 400.0;
  g_rMinBagSize_RS15_mm : REAL := 105.0;
  g_rMaxBagSize_RS26_mm : REAL := 760.0;
  g_rMinBagSize_RS26_mm : REAL := 160.0;
  g_rMaxBagSize_EnvB_mm : REAL := 760.0;
  g_rMinBagSize_EnvB_mm : REAL := 240.0;
END_VAR

VAR RETAIN
  g_rSizeEnvBPerf_mm : REAL := 520.0; (*Perimeter of the Envelope Bag Perf, in mm*)
END_VAR

VAR RETAIN
	gr_rMachMaxSpeed_BPM        : REAL := 1000.0; (*Parameter : machine max speed, in Bag/min*)
	gr_rHoldAxContactZone       : REAL := 22.0;   (*Parameter : zone where Holding Axis is in contact, in Deg*)
	gr_rTearAxContactZone       : REAL := 52.0;   (*Parameter : zone where Tearing Axis is in contact with the Bag, in Deg*)
	gr_rDrumAxContactZone       : REAL := 50.0;   (*Parameter : zone where Drum Axis is in contact with the blade, in Deg*)
	gr_rEnvBAxContactZone       : REAL := 26.0;   (*Parameter : zone where Envelope Bag Axis is in contact with the Bag, in Deg*)
	gr_rTearEBAxContactZone     : REAL := 52.0;   (*Parameter : zone where Tearing of the Envelope Bag Axis is in contact with the Bag, in Deg*)
	gr_rPosHoldBag              : REAL := 11.0;   (*Position of the Holding axis when the shaft is vertical, the bag is maintained, in°*)
	gr_rPosTearBag              : REAL := 26.0;   (*Position of the Tearing axis when the shaft is vertical, the bag is Teared, in°*)
	gr_rPosGripBag              : REAL := 25.0;   (*Position of the Drum axis when the blade is in the gripper, the bag is gripped, in°*)
	gr_rPosEnvBHoldBag          : REAL := 355.0;  (*Position of the Envelope Bag axis when the shaft is vertical, the bag is maintained and the nidles are outside, in°*)
	gr_rPosTearEBTearBag        : REAL := 18.0;   (*Position of the Tearing Envelope Bag axis when the shaft is vertical, the bag is Teared, in°*)
	gr_rAxisTimSet_SP_Vel       : REAL := 12;     (*Set point Velocity for Axis manual timing setting cycle, in Axis round/min*)
	gr_rAxisTimSet_SP_Acc       : REAL := 1200;   (*Set point Acceleration for Axis manual timing setting cycle, in Axis round/min²*)
	gr_rAxisTimSet_SP_Dec       : REAL := 3000;   (*Set point Deceleration for Axis manual timing setting cycle, in Axis round/min²*)
	gr_rMaxRangeWebDraw         : REAL := 1;      (*Max range for web draw modification on pull roll, in %*)
	gr_rLimOffsetRunVal         : REAL := 0.1;    (*Limit the max value of Offset changing when Running, in % of the Repeat*)
	gr_rIncrOffsetAxeRun        : REAL := 1.0;    (*Increment offset axis changing when Running, in mm/bag*)
	gr_tJogHornDur              : TIME := T#1s;   (*Horn duration in Jog, in s*)
	gr_tRunHornDur              : TIME := T#1s500ms; (*Horn duration in Run, in s*)
  gr_rMaxLSFlexoP_mmin        : REAL := 300.0; (*Max possible Line Speed with Flexo Press, in m/min*)
  gr_rDistPerfTearEnvBOn_mm   : REAL := 4560.0 ; (*4560.0 = Special distance for machine RS26_Pyrollpack_14661      Distance between position 0° Perf and Tearing for Envelope Bag case On, in mm*)
  gr_rDistPerfTearEnvBOff4_mm : REAL := 4260.0; (*4560.0+60.0 = Special distance for machine RS26_Pyrollpack_14661      Distance between position 0° Perf and Tearing for Envelope Bag case Off bags 2 grippers, in mm*)
  gr_rDistPerfTearEnvBOff2_mm : REAL := 4560.0; (*4560.0 = Special distance for machine RS26_Pyrollpack_14661       Distance between position 0° Perf and Tearing for Envelope Bag case Off bags 4 grippers, in mm*)
	gr_rSizeEnvBLowRol_mm       : REAL := 440.0;  (*Perimeter of the lower roller of the Envelope Bage Station = 140xpi, in mm*)
	gr_rTearCarStep_mm          : REAL := 413.0;  (*Step distance of tearing belts carriage. 1 rev of top roller of tearing station case 4 grippers on Drum = (39+2x1)xpi +2x1 because of belts thickness, in mm*)
	gr_rDistPerfTearRS26_mm     : REAL := 3800.0; (*Distance between position 0° Perf and Tearing for RS26 and without slitting in entry, in mm*)
	gr_rDistPerfTearRS15_mm     : REAL := 3700.0; (*Distance between position 0° Perf and Tearing for RS15 and without slitting in entry, in mm*)
	gr_rIncrShiftPerf_mm        : REAL := 1.0;    (*Increment shifting Perf in run, in mm*)
	gr_rBagSize2_4Hold_mm       : REAL := 160.0;  (*Bag size under which there are 4 tools on the holding, in mm*)
	gr_rBagSize1_2Hold_mm       : REAL := 320.0;  (*In case Envelope Bag size under which there are 2 tools on the holding instead of 1, in mm*)
	gr_rBagSize4_2Pliers_mm     : REAL := 400.0;  (*Bag size over which there are 2 pliers on the Drum, in mm*)
	gr_rEnvBSizeTear2_1_mm      : REAL := 500.0;  (*Envelope Bag, bag size over which tearing bag on the first Teraing Axis, in mm*)
	gr_rHMPerfSlowRot_rpm       : REAL := 2.0;    (*Slow Rotation speed of Hot Micro Perf Tool, in rpm*)
	gr_rHMPerfAcc_rpm2          : REAL := 120.0;  (*Acceleration Slow Rotation speed of Hot Micro Perf Tool, in rpm²*)
	gr_rHMPerfDec_rpm2          : REAL := 5000.0; (*Deceleration Slow Rotation speed of Hot Micro Perf Tool, in rpm²*)
	gr_rHMPerfSLActTool_mmin    : REAL := 20.0;   (*Line Speed Hot Micro Perf Tool activation, in m/min*)
	gr_bSetSpeedMode            : BOOL; (*Set Speed Mode =0:Auto, =1:Manu*)
END_VAR
VAR
	New_Variable : USINT := 0;
  gNormalStopReq : BOOL ;
  g_bBypassGuard : BOOL ;
	g_bTest_ : ARRAY[0..14] OF BOOL;
	g_iTest_ : ARRAY[0..14] OF INT;
	g_uiTest_ : ARRAY[0..14] OF UINT;
	g_iiTest_ : ARRAY[0..14] OF DINT;
	g_rTest_ : ARRAY[0..14] OF REAL;
END_VAR
VAR RETAIN
	g_bSim : BOOL;
END_VAR
```

### Program Logical/BagMachine_Section/3Web_Unit

#### 3Web_UnitCyclic.st
```iecst
(********************************************************************
 * COPYRIGHT -- .
 ********************************************************************
 * Program: 3Web_Unit
 * File: 3Web_UnitCyclic.st
 * Author: dominique
 * Created: November 05, 2011
 ********************************************************************
 * Implementation of program 3Web_Unit
 ********************************************************************)

PROGRAM _CYCLIC

// 3Web_Unit Fan On/Off
  gQ_CR_3W_Fan := gI_SS_3W_FanOnOff AND
                  NOT(g_bIndEStop)  AND
                  1                 ;

END_PROGRAM
```

#### 3Web_UnitInit.st
```iecst
(********************************************************************
 * COPYRIGHT -- .
 ********************************************************************
 * Program: 3Web_Unit
 * File: 3Web_UnitInit.st
 * Author: dominique
 * Created: November 05, 2011
 ********************************************************************
 * Implementation of program 3Web_Unit
 ********************************************************************)

PROGRAM _INIT

// Deflector Fan On/Off PB Colors
  HGW_2StatePB_0.BackColor_State0 := gBlue;
  HGW_2StatePB_0.ForeColor_State0 := gWhite;
  HGW_2StatePB_0.BackColor_State1 := gGreen;
  HGW_2StatePB_0.ForeColor_State1 := gBlack;

END_PROGRAM
```

### BagBundler.var - Global variables
```iecst
(********************************************************************
 * COPYRIGHT -- .
 ********************************************************************
 * Package: BagBundler
 * File: BagBundler.var
 * Author: dominique
 * Created: August 15, 2011
 ********************************************************************
 * Variables of package BagBundler
 ********************************************************************)

VAR
  g_bIndSelBundProd   : BOOL ;
  g_bIndBundManu      : BOOL ;
  g_bBundPackCountOK  : BOOL ;
  g_bIndBundReady     : BOOL ;
  g_bBundGuard_OK     : BOOL ;
  g_bBundJamFault     : BOOL ;
  g_bBundDriveFault   : BOOL ;
  g_bBundInitSep_OK   : BOOL ;
  g_bBundInitTilt_OK  : BOOL ;
  g_bBundInit_OK      : BOOL ;
  g_bBundAlarm_OK     : BOOL ;
  g_bBund_ManOn       : BOOL ;
  g_bBund_InitSep     : BOOL ;
  g_bBundStopInitSep  : BOOL ;
  g_bBund_InitTilt    : BOOL ;
  g_bBundStopInitTilt : BOOL ;
  g_bBund_InitHorn    : BOOL ;
  g_bBund_EndTravUp   : BOOL ;
  g_bBund_EndTravDown : BOOL ;
  g_bBund_SensFaultCycSep    : BOOL ; (*Sensor fault in Separator Cycle on Bundler*)
  g_bBund_SensFaultCycTilt   : BOOL ; (*Sensor fault in Tilter Cycle on Bundler*)
  g_bBund_SensorFault        : BOOL ; (*Sensor fault on Bundler*)
  g_bBund_TimOutFaultCycSep  : BOOL ;
  g_bBund_TimOutFaultCycTilt : BOOL ;
  g_bBund_TimOutFault        : BOOL ;
  g_bBund_MoveInSep_OK       : BOOL ;
  g_bBund_ResetCountReq      : BOOL ;
  g_bBund_StartTilt          : BOOL ;
  g_bBund_IndSpeedLimit      : BOOL ;

  g_tBund_TpWatchSens : TIME ;

  gHMI_Bund_SetPosTilt14C4InPB  : BOOL ;
  gHMI_Bund_SetPosTilt14C4OutPB : BOOL ;

END_VAR

VAR RETAIN
  gr_rPosTiltOffset0     : REAL := 0.95 ; (*Offset for setting position 0 of Tilter, in °*)
  gr_rPosTiltZLSpeed     : REAL := 15 ;   (*Low speed zone for Tilter motion, in°*)
  gr_rPosTiltTravel      : REAL := 60.0 ; (*Angle travel of Tilter, in °*)
  gr_rPosTiltStopUp      : REAL := 60.0 ; (*Pos stop Tilt up, in °*)
  gr_rPosTiltStopDown    : REAL := 2.0 ;  (*Pos stop Tilt down, in °*)
  gr_rPosTilt14C4In      : REAL := 1.0 ;  (*Tilter position for moving in cylinder 14C4, in °*)
  gr_rPosTiltTrav14C4Out : REAL := 52.0 ; (*Travel for moving out cylinder 14C4, in °*)
  gr_rMaxCyclPerMin      : REAL := 8.0 ;  (*Bundler maximum cycle per min, in Cycle/min*)

  gHMI_Bund_iBagCountStartTilt : INT ;
END_VAR

VAR
  gI_Bund_DriveFault : BOOL;
  gI_Bund_S106 : BOOL; (*Tilter end travel Down*)
  gI_Bund_S108 : BOOL; (*Tilter end travel Up*)
  gI_Bund_S103 : BOOL;
  gI_Bund_S101 : BOOL;
  gI_Bund_S102 : BOOL;
  gI_Bund_S109 : BOOL; (*Bundler Jam sensor*)
  gI_Bund_S104 : BOOL;
  gI_Bund_S110 : BOOL;
  gI_Bund_S111 : BOOL;
  gI_Bund_S112 : BOOL;
  gI_Bund_SpI1 : BOOL;
  gI_Bund_SpI2 : BOOL;
  gI_Bund_SpI3 : BOOL;
  gI_Bund_SpI4 : BOOL;
  gI_Bund_SafetyGuard : BOOL;
  gI_GSW_Bund         : BOOL;
  gI_Bund_EStopPB     : BOOL;
  gI_Bund_SlowerPB    : BOOL;
  gI_Bund_JogPB       : BOOL;
  gI_Bund_Stop        : BOOL;
  gAI_Bund_TiltPos    : INT;
  gQ_Bund_DriveStart  : BOOL;
  gQ_Bund_DriveDirection : BOOL;
  gQ_Bund_DriveFastSpeed : BOOL;
  gQ_Bund_DriveFailReset : BOOL;
  gQ_Bund_SOL_14C3Out : BOOL;
  gQ_Bund_SOL_14C4Out : BOOL;
  gQ_Bund_SOL_14C1Out : BOOL;
  gQ_Bund_SOL_14C2Out : BOOL;
  gQ_Bund_SOL_15C1Out : BOOL;
  gQ_Bund_SOL_AirSupply  : BOOL ;
  gQ_Bund_MotorBrake     : BOOL ;
  gQ_Bund_SOL_14C5Out    : BOOL;
  gQ_Bund_SOL_PresSelect : BOOL; (* Solenoid for selection of pressure of the cylinder contre-weight separator*)
  gQ_Bund_SpO3           : BOOL;
  gQ_Bund_SpO4           : BOOL;
  gQ_Bund_SpO5           : BOOL;

END_VAR

VAR CONSTANT

END_VAR
```

### Program Logical/BagMachine_Section/BagBundler/Control (IEC) - A new program

#### ControlCyclic.st - Cyclic code
```iecst
(********************************************************************
 * COPYRIGHT -- .
 ********************************************************************
 * Program: Control
 * File: ControlCyclic.st
 * Author: dominique
 * Created: August 16, 2011
 ********************************************************************
 * Implementation of program Control
 ********************************************************************)

PROGRAM _CYCLIC

    // -----------------------------------------------------------------
    // Control Bundler On
    IF bHMI_Bund_OnOff         AND
       NOT(gA[9].Ind_InMotion) AND
       NOT(g_bIndSelBundProd)  AND
       1                       THEN
      g_bIndSelBundProd := 1 ;
    END_IF
    // Control Bundler Off
    IF NOT(bHMI_Bund_OnOff)    AND
       NOT(gA[9].Ind_InMotion) AND
       g_bIndSelBundProd       AND
       1                       THEN
      g_bIndSelBundProd := 0 ;
    END_IF

    // -----------------------------------------------------------------
    // Control local Bundler manu mode
    bBundManOn  := EDGEPOS(bHMI_Bund_ManOn_PB) AND NOT(g_bIndBundManu) ;
    bBundManOff := EDGEPOS(bHMI_Bund_ManOn_PB) AND g_bIndBundManu ;
    // On
    IF bBundManOn              AND
       gManualMode_On          AND
       NOT(gA[9].Ind_InMotion) AND
       1                       THEN
      g_bIndBundManu := 1 ;
      iHMI_BundManLock := 1 ;
    END_IF
    // Off
    IF ( bBundManOff           OR
         NOT(gManualMode_On) ) AND
       1                       THEN
      g_bIndBundManu := 0 ;
      iHMI_BundManLock := 0 ;
    END_IF

    //Manu Mode Off/On From HMI
      H_FB_ToggleTB_0.IN_bTB := g_bIndBundManu ;
      uiBundManTxt_Ind  := H_FB_ToggleTB_0.OUT_uiTxt_Ind;
      uiBundManCol_Ind  := H_FB_ToggleTB_0.OUT_uiCol_Ind;
      H_FB_ToggleTB_0();

    // -----------------------------------------------------------------
    // Guards
    g_bBundGuard_OK := 1 ; //NOT(gI_GSW_Bund) OR g_bIndSelBundProd ;   D.M. 03/08/2011 BrownPaper_14542 Not used on this machine

    // -----------------------------------------------------------------
    // Bundler ready
    g_bIndBundReady := g_bBundAlarm_OK        AND
                       g_bBundInit_OK         AND
                       NOT(g_bIndBundManu)    OR
                       NOT(g_bIndSelBundProd) AND
                       1                      ;

    // -----------------------------------------------------------------
    // General alarme on Bundler
    g_bBundAlarm_OK := g_bBundGuard_OK                 AND
                       NOT(g_bBundDriveFault)          AND
                       NOT(g_bBundJamFault)            AND
                       NOT(g_bBund_SensorFault)        AND
                       NOT(g_bBund_TimOutFault)        OR
                       NOT(g_bIndSelBundProd)          AND
                       1                               ;

    // Reset init indicator in case of fault
    IF NOT(g_bBundAlarm_OK) OR
       g_bIndBundManu       THEN
      g_bBundInitSep_OK  := 0 ;
      g_bBundInitTilt_OK := 0 ;
    END_IF ;
    g_bBundInit_OK := g_bBundInitSep_OK AND g_bBundInitTilt_OK OR NOT(g_bIndSelBundProd) ;

    // Air suply
    gQ_Bund_SOL_AirSupply := g_bBundGuard_OK           AND
                             gBagMachine_EstopAlarmsOK AND
                             g_bIndSelBundProd         AND
                             g_bMainPower_On           AND
                             1                         ;

    // Sensor fault
    g_bBund_SensorFault := g_bBund_SensFaultCycSep OR g_bBund_SensFaultCycTilt ;
    // Step Time out
    g_bBund_TimOutFault := g_bBund_TimOutFaultCycTilt OR g_bBund_TimOutFaultCycSep ;

    // Reset cycle and sensor fault
    IF EDGEPOS(gAlarmReset) THEN
      g_bBund_SensFaultCycSep    := 0 ;
      g_bBund_SensFaultCycTilt   := 0 ;
      g_bBund_TimOutFaultCycSep  := 0 ;
      g_bBund_TimOutFaultCycTilt := 0 ;
    END_IF ;

    // ------------------------------------------------------------------
    // Init Bundler
    // Permissive
    bBundInit_Perm := NOT(gA[9].Ind_InMotion) AND
                      g_bBundAlarm_OK         AND
                      g_bIndSelBundProd       AND
                      NOT(g_bBundDriveFault)  AND
                      1                       ;
    // Start cycle
    bInitBundStart := bHMI_Bund_Init_PB AND NOT(bInitBund) AND NOT(stTP_0.Q) ;
    // Stop cycle
    IF EDGEPOS(bHMI_Bund_Init_PB) AND
       bInitBund                  THEN
      bInitBundStop := 1 ;
      g_bBundStopInitSep  := 1 ;
      g_bBundStopInitTilt := 1 ;
    END_IF
    stTP_0(IN:=bInitBundStop, PT:=T#2s) ;
    IF NOT(stTP_0.Q) THEN
      bInitBundStop := 0 ;
    END_IF

    H_FB_2StepMove_0.IN_bStart  := bInitBundStart ;
    H_FB_2StepMove_0.IN_bPermis := bBundInit_Perm ;
    H_FB_2StepMove_0.IN_tTpHorn := tBundInitTpHorn ;
    H_FB_2StepMove_0();
    g_bBund_InitHorn := H_FB_2StepMove_0.OUT_bHorn ;

    IF EDGEPOS(H_FB_2StepMove_0.OUT_bStartMove) AND
       1                                        THEN
      g_bBund_InitSep  := 1 ;
      g_bBund_InitTilt := 1 ;
      g_bBund_SensFaultCycSep    := 0 ;
      g_bBund_SensFaultCycTilt   := 0 ;
      g_bBund_TimOutFaultCycSep  := 0 ;
      g_bBund_TimOutFaultCycTilt := 0 ;
    END_IF
    bInitBund := g_bBund_InitSep  OR
                 g_bBund_InitTilt ;

    // Init button HMI display
    CASE H_FB_2StepMove_0.OUT_iActStep OF
      1 : // Horn ringing
          uiBundInitTxt_Ind := 1 ;
          uiBundInitCol_Ind := gGreen + gBlack * 256 ;
      2..3 : // Waiting remove start
          uiBundInitTxt_Ind := 1 ;
          uiBundInitCol_Ind := gBlue + gWhite * 256 ;
      4 : // New start OK
          uiBundInitTxt_Ind := 1 ;
          uiBundInitCol_Ind := gGreen + gBlack * 256 ;
    ELSE
      IF NOT(bInitBund) THEN
        // Waiting start
        uiBundInitTxt_Ind := 0 ;
        uiBundInitCol_Ind := gBlue + gWhite * 256 ;
      ELSE
        // Cycle running
        uiBundInitTxt_Ind := 2 ;
        uiBundInitCol_Ind := gRed + gBlack * 256 ;
      END_IF ;
    END_CASE ;

END_PROGRAM
```

### Program Logical/BagMachine_Section/BagBundler/Separator (IEC) - A new program

#### Separator.var
```iecst
(********************************************************************
 * COPYRIGHT -- .
 ********************************************************************
 * Program: Separator
 * File: Separator.var
 * Author: dominique
 * Created: August 15, 2011
 ********************************************************************
 * Local variables of program Separator
 ********************************************************************)

VAR
  stCycBundSep        : CycGen ;
  bQ_Bund_SOL_14C1Out : BOOL;
  bQ_Bund_SOL_14C2Out : BOOL;
  bQ_Bund_SOL_PresSelect : BOOL;

  stTON_RetCyl14C1 : TON ;
  tTpRetCyl14C1    : TIME ;
  bInitSepCycl     : BOOL ;
  stTON_WatchCyc   : TON ;
  tTpWatchCyc      : TIME ;
  iMemoStepCyc     : INT ;
  stTON_SelPres    : TON ;

  bHMI_BundMan_14C1P_PB   : BOOL ;
  bHMI_BundMan_14C1M_PB   : BOOL ;
  iHMI_Bund_14C1In_State  : INT ;
  iHMI_Bund_14C1Out_State : INT ;
  bHMI_BundMan_14C2P_PB   : BOOL ;
  bHMI_BundMan_14C2M_PB   : BOOL ;
  iHMI_Bund_14C2In_State  : INT ;
  iHMI_Bund_14C2Out_State : INT ;
  bHMI_BundMan_PresSelect_PB : BOOL ;
  iHMI_Bund_S101 : INT ;
  iHMI_Bund_S102 : INT ;
  iHMI_Bund_S103 : INT ;
  iHMI_Bund_S109 : INT ;

  bS101_FaultIn  : BOOL ;
  bS101_FaultOut : BOOL ;
  bS101_Fault    : BOOL ;
  bS102_FaultIn  : BOOL ;
  bS102_FaultOut : BOOL ;
  bS102_Fault    : BOOL ;

  H_FB_WS_14C1 : H_FB_WatchSensor ;
  H_FB_WS_14C2 : H_FB_WatchSensor ;

  H_FB_Flash_0 : H_FB_Flash ;
  bFlash : BOOL ;

  HGW_2StatePB_0 : HGW_2StatePB ;
  uiPresSelPBTxt_Id : UINT ;
  uiPresSelPBCol_Id : UINT ;

  iTest : INT ;
  stCycBundTilt : CycGen;
  tTpSelPres : TIME;
END_VAR

VAR CONSTANT

END_VAR
```

### Program Logical/BagMachine_Section/BagBundler/Tilter (IEC) - A new program

#### Tilter.var
```iecst
(********************************************************************
 * COPYRIGHT -- .
 ********************************************************************
 * Program: Tilting
 * File: Tilting.var
 * Author: dominique
 * Created: August 16, 2011
 ********************************************************************
 * Local variables of program Tilting
 ********************************************************************)

VAR
  stCycBundTilt          : CycGen ;
  bQ_Bund_DriveStart     : BOOL;
  bQ_Bund_DriveDirection : BOOL;
  bQ_Bund_DriveFastSpeed : BOOL;
  bQ_Bund_SOL_14C3Out    : BOOL;
  bQ_Bund_SOL_14C4Out    : BOOL;
  bQ_Bund_SOL_14C5Out    : BOOL;

  rPosTiltUpLSpeed   : REAL ;
  rPosTiltDownLSpeed : REAL ;
  rPosTiltUpStop     : REAL ;
  rPosTiltDownStop   : REAL ;
  rPosTiltDegPts     : REAL ; (*Conversion AI points in degrees for Tilter position, in Deg/pts*)

  bHMI_Cmd_RecPosIn14C1 : BOOL ;
  rHMI_PosTiltAct  : REAL ;
  rK_HMI : REAL ;

  bHMI_BundMan_14C3P_PB   : BOOL ;
  bHMI_BundMan_14C3M_PB   : BOOL ;
  iHMI_Bund_14C3In_State  : INT ;
  iHMI_Bund_14C3Out_State : INT ;
  bHMI_BundMan_14C4P_PB   : BOOL ;
  bHMI_BundMan_14C4M_PB   : BOOL ;
  iHMI_Bund_14C4In_State  : INT ;
  iHMI_Bund_14C4Out_State : INT ;
  bHMI_BundMan_14C5P_PB   : BOOL ;
  bHMI_BundMan_14C5M_PB   : BOOL ;
  iHMI_Bund_14C5In_State  : INT ;
  iHMI_Bund_14C5Out_State : INT ;
  bHMI_BundMan_TiltUp_PB   : BOOL;  (*Manu move up tilter*)
  bHMI_BundMan_TiltDown_PB : BOOL;  (*Manu move down tilter*)
  iHMI_Bund_S104 : INT ;
  iHMI_Bund_S106 : INT ;
  iHMI_Bund_S108 : INT ;
  iHMI_Bund_S110 : INT ;
  iHMI_Bund_S111 : INT ;
  iHMI_Bund_S112 : INT ;
  iHMI_Bund_EndTravUp   : INT ;
  iHMI_Bund_EndTravDown : INT ;

  bS104_FaultIn  : BOOL ;
  bS104_FaultOut : BOOL ;
  bS104_Fault    : BOOL ;
  bS110_FaultIn  : BOOL ;
  bS110_FaultOut : BOOL ;
  bS110_Fault    : BOOL ;
  bS111_FaultIn  : BOOL ;
  bS111_FaultOut : BOOL ;
  bS111_Fault    : BOOL ;
  bS112_FaultIn  : BOOL ;
  bS112_FaultOut : BOOL ;
  bS112_Fault    : BOOL ;

  H_FB_WS_14C3 : H_FB_WatchSensor ;
  H_FB_WS_14C4 : H_FB_WatchSensor ;
  H_FB_WS_14C5 : H_FB_WatchSensor ;

  bIndLSpeed      : BOOL ;
  bIndPosUpStop   : BOOL ;
  bIndPosDownStop : BOOL ;

  rPosTiltAct      : REAL ;
  rPosTiltActTemp1 : REAL ;
  rMemoPosTiltActTemp1 : REAL ;
  rMemoPosTiltAct  : REAL ;
  rNumRoundTilt    : REAL ;
  bMoveTiltPos     : BOOL ;
  rPosTiltActTemp2 : REAL ;
  rPosTiltActTemp3 : REAL ;
  rPosTiltActTemp4 : REAL ;
  iCmpt            : INT ;
  rK               : REAL ; (*Tilter postion filtering factor*)
  rPosTiltInit_OK  : REAL ; (*Position threshold for Tilter in position init OK, in °*)
  rPosTiltInitHyst : REAL ;
  bPosTiltInit_OK  : BOOL ;
  stTON_StopTilt   : TON ;
  bTON_StopTilt_IN : BOOL ;
  tTpStopTilt      : TIME ;
  bInitTiltCycl    : BOOL ;
  stTON_Out14C5    : TON ;
  tTpOut14C5       : TIME ;
  stTON_Out14C3    : TON ;
  tTpOut14C3       : TIME ;
  stTON_WatchCyc   : TON ;
  tTpWatchCyc      : TIME ;
  iMemoStepCyc     : INT ;

  H_FB_Flash_0 : H_FB_Flash ;
  bFlash : BOOL ;

  rPosTilt14C4Out : REAL;
  TESTTILT : BOOL;
  starttilter_without_S103 : BOOL;
END_VAR

VAR CONSTANT

END_VAR
```

#### TilterCyclic.st
```iecst
(********************************************************************
 * COPYRIGHT -- .
 ********************************************************************
 * Program: Tilter
 * File: TilterCyclic.st
 * Author: dominique
 * Created: August 16, 2011
 ********************************************************************
 * Implementation of program Tilter
 ********************************************************************)

PROGRAM _CYCLIC

    // End travel Tilter
    g_bBund_EndTravUp   := gI_Bund_S108 AND bQ_Bund_DriveDirection AND bQ_Bund_DriveStart ;
    g_bBund_EndTravDown := gI_Bund_S106 AND NOT(bQ_Bund_DriveDirection) AND bQ_Bund_DriveStart ;

    // Output assignments
    gQ_Bund_SOL_14C3Out := bQ_Bund_SOL_14C3Out AND gBagMachine_EstopAlarmsOK ;
    gQ_Bund_SOL_14C4Out := bQ_Bund_SOL_14C4Out AND gBagMachine_EstopAlarmsOK ;
    gQ_Bund_SOL_14C5Out := bQ_Bund_SOL_14C5Out AND gBagMachine_EstopAlarmsOK ;

    // Drive Tilter
    gQ_Bund_DriveStart := bQ_Bund_DriveStart AND gBagMachine_EstopAlarmsOK    AND
                          NOT(g_bBund_EndTravUp) AND NOT(g_bBund_EndTravDown) ;
    gQ_Bund_DriveDirection := bQ_Bund_DriveDirection AND gBagMachine_EstopAlarmsOK AND
                              NOT(g_bBund_EndTravUp) AND NOT(g_bBund_EndTravDown)  ;
    gQ_Bund_DriveFastSpeed := bQ_Bund_DriveFastSpeed AND gBagMachine_EstopAlarmsOK AND
                              NOT(g_bBund_EndTravUp) AND NOT(g_bBund_EndTravDown)  ;
    gQ_Bund_DriveFailReset := gAlarmReset ;

    gQ_Bund_MotorBrake := gQ_Bund_DriveStart OR gQ_Bund_DriveFastSpeed ;

    //---------------------------------------------------------------------------------------------------------------------
    // Sensor watching

    H_FB_Flash_0(IN_bEnable:=1, IN_rNumFlashPerSec:=2) ;
    bFlash := H_FB_Flash_0.OUT_bFlash ;

    // S104 on 14C3 In
    H_FB_WS_14C3.IN_bSensorIn   := gI_Bund_S104 ;
    H_FB_WS_14C3.IN_bSOL_In     := NOT(gQ_Bund_SOL_14C3Out) ;
    H_FB_WS_14C3.IN_bSOL_Out    := gQ_Bund_SOL_14C3Out ;
    H_FB_WS_14C3.IN_bActSensIn  := 1 ;
    H_FB_WS_14C3.IN_bActSensOut := 0 ;
    H_FB_WS_14C3.IN_tTpWatchIn  := g_tBund_TpWatchSens ;
    H_FB_WS_14C3.IN_tTpWatchOut := g_tBund_TpWatchSens ;
    H_FB_WS_14C3.IN_bReset      := gAlarmReset ;
    H_FB_WS_14C3();
    bS104_FaultOut := H_FB_WS_14C3.OUT_bSensIn_FaultOut ;
    bS104_FaultIn  := H_FB_WS_14C3.OUT_bSensIn_FaultIn ;
    bS104_Fault    := H_FB_WS_14C3.OUT_bSensIn_Fault ;

    // S110 on 14C4 In
    H_FB_WS_14C4.IN_bSensorIn   := gI_Bund_S110 ;
    H_FB_WS_14C4.IN_bSOL_In     := NOT(gQ_Bund_SOL_14C4Out) ;
    H_FB_WS_14C4.IN_bSOL_Out    := gQ_Bund_SOL_14C4Out ;
    H_FB_WS_14C4.IN_bActSensIn  := 1 ;
    H_FB_WS_14C4.IN_bActSensOut := 0 ;
    H_FB_WS_14C4.IN_tTpWatchIn  := g_tBund_TpWatchSens ;
    H_FB_WS_14C4.IN_tTpWatchOut := g_tBund_TpWatchSens ;
    H_FB_WS_14C4.IN_bReset      := gAlarmReset ;
    H_FB_WS_14C4();
    bS110_FaultOut := H_FB_WS_14C4.OUT_bSensIn_FaultOut ;
    bS110_FaultIn  := H_FB_WS_14C4.OUT_bSensIn_FaultIn ;
    bS110_Fault    := H_FB_WS_14C4.OUT_bSensIn_Fault ;

    // S111 and S112 on 14C5 In and Out
    H_FB_WS_14C5.IN_bSensorIn   := gI_Bund_S111 ;
    H_FB_WS_14C5.IN_bSensorOut  := gI_Bund_S112 ;
    H_FB_WS_14C5.IN_bSOL_In     := NOT(gQ_Bund_SOL_14C5Out) ;
    H_FB_WS_14C5.IN_bSOL_Out    := gQ_Bund_SOL_14C5Out ;
    H_FB_WS_14C5.IN_bActSensIn  := 1 ;
    H_FB_WS_14C5.IN_bActSensOut := 1 ;
    H_FB_WS_14C5.IN_tTpWatchIn  := g_tBund_TpWatchSens ;
    H_FB_WS_14C5.IN_tTpWatchOut := g_tBund_TpWatchSens ;
    H_FB_WS_14C5.IN_bReset      := gAlarmReset ;
    H_FB_WS_14C5();
    bS111_FaultOut := H_FB_WS_14C5.OUT_bSensIn_FaultOut ;
    bS111_FaultIn  := H_FB_WS_14C5.OUT_bSensIn_FaultIn ;
    bS111_Fault    := H_FB_WS_14C5.OUT_bSensIn_Fault ;
    bS112_FaultOut := H_FB_WS_14C5.OUT_bSensOut_FaultOut ;
    bS112_FaultIn  := H_FB_WS_14C5.OUT_bSensOut_FaultIn ;
    bS112_Fault    := H_FB_WS_14C5.OUT_bSensOut_Fault ;

    // HMI Sensors states display
    IF gI_Bund_S104 THEN
      iHMI_Bund_S104 := 1 ;
    ELSE
      iHMI_Bund_S104 := 0 ;
    END_IF
    IF bS104_Fault AND
       bFlash      THEN
      iHMI_Bund_S104 := 2 ;
    END_IF

    IF gI_Bund_S106 THEN
      iHMI_Bund_S106 := 1 ;
      IF g_bBund_EndTravDown AND
         bFlash              THEN
        iHMI_Bund_S106 := 2 ;
      END_IF
    ELSE
      iHMI_Bund_S106 := 0 ;
    END_IF

    IF gI_Bund_S108 THEN
      iHMI_Bund_S108 := 1 ;
      IF g_bBund_EndTravUp AND
         bFlash            THEN
        iHMI_Bund_S108 := 2 ;
      END_IF
    ELSE
      iHMI_Bund_S108 := 0 ;
    END_IF

    IF gI_Bund_S110 THEN
      iHMI_Bund_S110 := 1 ;
    ELSE
      iHMI_Bund_S110:= 0 ;
    END_IF
    IF bS110_Fault AND
       bFlash      THEN
      iHMI_Bund_S110 := 2 ;
    END_IF

    IF gI_Bund_S111 THEN
      iHMI_Bund_S111 := 1 ;
    ELSE
      iHMI_Bund_S111 := 0 ;
    END_IF
    IF bS111_Fault AND
       bFlash      THEN
      iHMI_Bund_S111 := 2 ;
    END_IF

    IF gI_Bund_S112 THEN
      iHMI_Bund_S112 := 1 ;
    ELSE
      iHMI_Bund_S112 := 0 ;
    END_IF
    IF bS112_Fault AND
       bFlash      THEN
      iHMI_Bund_S112 := 2 ;
    END_IF

    g_bBund_SensFaultCycTilt := bS104_Fault OR bS110_Fault OR bS111_Fault OR bS112_Fault ;

    // HMI Cylinders states display
    // Cylinder 14C3
    // Case Out
    IF gQ_Bund_SOL_14C3Out THEN
      iHMI_Bund_14C3Out_State := 1 ;
      iHMI_Bund_14C3In_State  := 0 ;
    END_IF
    IF bS104_FaultOut THEN
      IF bFlash THEN
        iHMI_Bund_14C3Out_State := 2 ;
      ELSE
        iHMI_Bund_14C3Out_State := 3 ;
      END_IF
    END_IF
    // Case In
    IF NOT(gQ_Bund_SOL_14C3Out) THEN
      iHMI_Bund_14C3In_State  := 4 ;
      iHMI_Bund_14C3Out_State := 0 ;
    END_IF
    IF bS104_FaultIn THEN
      IF bFlash THEN
        iHMI_Bund_14C3In_State := 5 ;
      ELSE
        iHMI_Bund_14C3In_State := 6 ;
      END_IF
    END_IF

    // Cylinder 14C4
    // Case Out
    IF gQ_Bund_SOL_14C4Out THEN
      iHMI_Bund_14C4Out_State := 4 ;
      iHMI_Bund_14C4In_State  := 0 ;
    END_IF
    IF bS110_FaultOut THEN
      IF bFlash THEN
        iHMI_Bund_14C4Out_State := 5 ;
      ELSE
        iHMI_Bund_14C4Out_State := 6 ;
      END_IF
    END_IF
    // Case In
    IF NOT(gQ_Bund_SOL_14C4Out) THEN
      iHMI_Bund_14C4In_State  := 1 ;
      iHMI_Bund_14C4Out_State := 0 ;
    END_IF
    IF bS110_FaultIn THEN
      IF bFlash THEN
        iHMI_Bund_14C4In_State := 2 ;
      ELSE
        iHMI_Bund_14C4In_State := 3 ;
      END_IF
    END_IF

    // Cylinder 14C5
    // Case Out
    IF gQ_Bund_SOL_14C5Out THEN
      iHMI_Bund_14C5Out_State := 1 ;
      iHMI_Bund_14C5In_State  := 0 ;
    END_IF
    IF bS111_FaultOut OR bS112_FaultOut THEN
      IF bFlash THEN
        iHMI_Bund_14C5Out_State := 2 ;
      ELSE
        iHMI_Bund_14C5Out_State := 3 ;
      END_IF
    END_IF
    // Case In
    IF NOT(gQ_Bund_SOL_14C5Out) THEN
      iHMI_Bund_14C5In_State  := 4 ;
      iHMI_Bund_14C5Out_State := 0 ;
    END_IF
    IF bS111_FaultIn OR bS112_FaultIn THEN
      IF bFlash THEN
        iHMI_Bund_14C5In_State := 5 ;
      ELSE
        iHMI_Bund_14C5In_State := 6 ;
      END_IF
    END_IF

     // --------------------------------------------------
     // HIM Tilter postion setup
     IF EDGEPOS(bHMI_Cmd_RecPosIn14C1) AND
        NOT(bQ_Bund_DriveStart)        THEN
       gr_rPosTilt14C4In := rPosTiltAct ;
     END_IF

     // --------------------------------------------------
     // Calculations
     rPosTiltUpLSpeed   := gr_rPosTiltTravel - gr_rPosTiltZLSpeed ;
     rPosTiltDownLSpeed := gr_rPosTiltZLSpeed ;
     rPosTiltUpStop     := gr_rPosTiltStopUp ;
     rPosTiltDownStop   := gr_rPosTiltStopDown ;

     // Tilter  actual position mesured
     rPosTiltActTemp1 := INT_TO_REAL(gAI_Bund_TiltPos) * rPosTiltDegPts + gr_rPosTiltOffset0 ;
     rPosTiltActTemp4 := gr_rPosTiltTravel - rPosTiltActTemp1 ;
     // Filtering mesured position (Lowpass PT1)
     rPosTiltActTemp2 := ( rPosTiltActTemp1 + rK * rPosTiltActTemp2 ) / ( rK + 1 ) ;
     rPosTiltActTemp3 := gr_rPosTiltTravel - rPosTiltActTemp2 ;

     IF (( rPosTiltActTemp4 - rMemoPosTiltAct ) < -10) AND
        bQ_Bund_DriveDirection                         THEN
       rNumRoundTilt := 1 ;
     END_IF
     IF (( rPosTiltActTemp4 - rMemoPosTiltAct ) > 10) AND
        NOT(bQ_Bund_DriveDirection)                   THEN
       rNumRoundTilt := 0 ;
     END_IF
     IF iCmpt > 10 THEN
       iCmpt := 0 ;
       rMemoPosTiltAct := rPosTiltActTemp4 ;
     END_IF
     iCmpt := iCmpt + 1 ;

     rPosTiltAct := rPosTiltActTemp3 + rNumRoundTilt * gr_rPosTiltTravel ;
     IF rPosTiltAct < 0.0 THEN
       rPosTiltAct := 0.0 ;
     END_IF

     // HMI display filtering
     rHMI_PosTiltAct := ( rPosTiltAct + rK_HMI * rHMI_PosTiltAct ) / ( rK_HMI + 1 )  ;
     IF rHMI_PosTiltAct < 0.0 THEN
       rHMI_PosTiltAct := 0.0 ;
     END_IF

     // Pos init Tilter OK
     IF rPosTiltAct <= rPosTiltInit_OK THEN
       bPosTiltInit_OK := 1 ;
     END_IF
     IF rPosTiltAct > (rPosTiltInit_OK + rPosTiltInitHyst) THEN
       bPosTiltInit_OK := 0 ;
     END_IF

     // Position Tilter for move out cylinder 14C4
     rPosTilt14C4Out := gr_rPosTilt14C4In + gr_rPosTiltTrav14C4Out ;

     // Tilter position indicator
     rPosTiltUpLSpeed   := rPosTiltUpStop - gr_rPosTiltZLSpeed ;
     rPosTiltDownLSpeed := rPosTiltDownStop + gr_rPosTiltZLSpeed ;
     // Low speed selection
     bIndLSpeed := ( rPosTiltAct >= rPosTiltUpLSpeed )   AND
                   bQ_Bund_DriveDirection                OR
                   ( rPosTiltAct <= rPosTiltDownLSpeed ) AND
                   NOT(bQ_Bund_DriveDirection)           OR
                   g_bIndBundManu                        ;

    IF ( rPosTiltAct >= rPosTiltUpStop ) OR
       gI_Bund_S108                      THEN
      bIndPosUpStop := 1 ;
    END_IF
    IF ( rPosTiltAct >= 20.0 )          AND
       ( rPosTiltAct < rPosTiltUpStop ) AND
       NOT(gI_Bund_S108)                THEN
      bIndPosUpStop := 0 ;
    END_IF
    IF ( rPosTiltAct <= rPosTiltDownStop ) OR
       gI_Bund_S106                        THEN
      bIndPosDownStop := 1 ;
    END_IF
    IF ( rPosTiltAct <= 40.0 )            AND
       ( rPosTiltAct > rPosTiltDownStop ) AND
       NOT(gI_Bund_S106)                  THEN
      bIndPosDownStop := 0 ;
    END_IF

    //---------------------------------------------------------------------------------------------------------------------
    // Tilter cycle
    //---------------------------------------------------------------------------------------------------------------------

    // Start cycle
    IF g_bIndSelBundProd               AND
       gBagMachine_EstopAlarmsOK       AND
       NOT(bInitTiltCycl)              AND
       NOT(g_bBund_SensFaultCycTilt)   AND
       NOT(g_bBund_TimOutFaultCycTilt) AND
       1                               THEN
      stCycBundTilt.bSCyc := 1 ;
    END_IF ;

    //----------------------------------------------------------------------
    // Cycle at rest
    IF NOT(stCycBundTilt.bSCyc) AND
       1                       THEN
      IF NOT( stCycBundTilt.bFCyc ) THEN
        // Init after cycle unpropaly ended
        stCycBundTilt.bFCyc := 1 ;
        stCycBundTilt.bCyc  := 0 ;
        stCycBundTilt.bCycFail := 1 ;

        bInitTiltCycl          := 0 ;
        g_bBund_InitTilt       := 0 ;
        bQ_Bund_DriveStart     := 0 ;
        bQ_Bund_DriveFastSpeed := 0 ;
        bQ_Bund_DriveDirection := 0 ;
      END_IF
      stCycBundTilt.iStep := 0 ;
      RETURN ;
    ELSE
    //----------------------------------------------------------------------
    // Cycle running

    // Manu mode
      IF g_bIndBundManu THEN
        stCycBundTilt.iStep := C_iSTEP_25 ;
        // In manu mode cycle is frozen in Step 25
        IF bHMI_BundMan_14C3P_PB THEN
          bQ_Bund_SOL_14C3Out := 1 ;
        END_IF
        IF bHMI_BundMan_14C3M_PB THEN
          bQ_Bund_SOL_14C3Out := 0 ;
        END_IF
        IF bHMI_BundMan_14C4P_PB THEN
          bQ_Bund_SOL_14C4Out := 1 ;
        END_IF
        IF bHMI_BundMan_14C4M_PB THEN
          bQ_Bund_SOL_14C4Out := 0 ;
        END_IF
        IF bHMI_BundMan_14C5P_PB THEN
          bQ_Bund_SOL_14C5Out := 1 ;
        END_IF
        IF bHMI_BundMan_14C5M_PB THEN
          bQ_Bund_SOL_14C5Out := 0 ;
        END_IF
        bQ_Bund_DriveStart     := bHMI_BundMan_TiltUp_PB OR bHMI_BundMan_TiltDown_PB ;
        bQ_Bund_DriveDirection := bHMI_BundMan_TiltUp_PB ;
      END_IF
      IF NOT(g_bIndBundManu) THEN
        bHMI_BundMan_14C3P_PB := 0 ;
        bHMI_BundMan_14C4P_PB := 0 ;
        bHMI_BundMan_14C5P_PB := 0 ;
        bHMI_BundMan_TiltUp_PB   := 0 ;
        bHMI_BundMan_TiltDown_PB := 0 ;
      END_IF

    // Permanent conditions
      IF NOT(gBagMachine_EstopAlarmsOK) OR
         g_bBund_SensFaultCycTilt       THEN
        stCycBundTilt.bSCyc := 0 ;
        bHMI_BundMan_14C3P_PB := 0 ;
        bHMI_BundMan_14C4P_PB := 0 ;
        bHMI_BundMan_14C5P_PB := 0 ;
        bHMI_BundMan_TiltUp_PB   := 0 ;
        bHMI_BundMan_TiltDown_PB := 0 ;
        bQ_Bund_DriveStart     := 0 ;
        bQ_Bund_DriveFastSpeed := 0 ;
        bQ_Bund_DriveDirection := 0 ;
      END_IF

      // Init cycle
      // Start init
      IF g_bBund_InitTilt   AND
         NOT(bInitTiltCycl) THEN
        bInitTiltCycl       := 1 ;
        g_bBundInitTilt_OK  := 0 ;
        // Put cycle in Step
        IF (rPosTiltAct >= rPosTilt14C4Out) THEN
          stCycBundTilt.iStep := C_iSTEP_15 ;
          // Action Step 15
          bQ_Bund_SOL_14C3Out := 1 ;
          bQ_Bund_SOL_14C4Out := 1 ;
        ELSE
          stCycBundTilt.iStep := C_iSTEP_4 ;
        // Action Step 4
          bQ_Bund_SOL_14C3Out    := 0 ;
          bQ_Bund_SOL_14C4Out    := 0 ;
          bQ_Bund_DriveStart     := 1 ;
          bQ_Bund_DriveDirection := 1 ;
          g_bBund_StartTilt      := 0 ;
          iMemoStepCyc           := C_iSTEP_99 ;
        END_IF
        // Init cycle
        stCycBundTilt.bFCyc := 0 ;
        stCycBundTilt.bCyc  := 1 ;
        stCycBundTilt.bCycFail := 0 ;
        g_bBund_MoveInSep_OK   := 0 ;
      END_IF
      // Stop init
      IF g_bBundStopInitTilt THEN
        g_bBund_InitTilt    := 0 ;
        g_bBundInitTilt_OK  := 0 ;
        g_bBundStopInitTilt := 0 ;
        stCycBundTilt.bSCyc := 0 ;
      END_IF

      // Watching Step time out
      IF g_bIndBundManu                      OR
         ( stCycBundTilt.iStep < C_iSTEP_4 ) THEN

        iMemoStepCyc := C_iSTEP_99 ;
        stTON_WatchCyc(IN:=(iMemoStepCyc=stCycBundTilt.iStep), PT:=tTpWatchCyc);
      ELSE
        stTON_WatchCyc(IN:=(iMemoStepCyc=stCycBundTilt.iStep), PT:=tTpWatchCyc);
        iMemoStepCyc := stCycBundTilt.iStep ;
      END_IF
      IF stTON_WatchCyc.Q THEN
        g_bBund_TimOutFaultCycTilt := 1 ;
        //stCycBundTilt.bSCyc := 0 ;
      END_IF

    // Permanent actions
      bTON_StopTilt_IN := ( (stCycBundTilt.iStep = C_iSTEP_7)  AND bIndPosUpStop     OR
                            (stCycBundTilt.iStep = C_iSTEP_11) AND bIndPosDownStop ) ;
      stTON_StopTilt (
            IN := bTON_StopTilt_IN ,
            PT := tTpStopTilt
                     ) ;

      // Tilter speed
      bQ_Bund_DriveFastSpeed := NOT(bIndLSpeed) AND bQ_Bund_DriveStart ;

      // Cylinder 14C5
      stTON_Out14C5(IN:=gI_Bund_S112 AND NOT(g_bIndBundManu), PT:=tTpOut14C5) ;
      IF stTON_Out14C5.Q THEN
        bQ_Bund_SOL_14C5Out := 0 ;
      END_IF

      // Cylinder 14C3
      stTON_Out14C3(IN:=bQ_Bund_SOL_14C3Out AND NOT(g_bIndBundManu), PT:=tTpOut14C3) ;

    END_IF
    //----------------------------------------------------------------------
    // Cycle steps

        CASE stCycBundTilt.iStep OF

        C_iSTEP_0 :
         //----------------------------------------------
         // Etape 1 : Initialisation cycle
         //----------------------------------------------
          IF TRUE THEN
            stCycBundTilt.iStep := C_iSTEP_1 ;

            // Action Step 1
            stCycBundTilt.bFCyc := 0 ;
            stCycBundTilt.bCyc  := 1 ;
            stCycBundTilt.bCycFail := 0 ;

            g_bBund_MoveInSep_OK := 0 ;
          END_IF

        C_iSTEP_1 :
         //----------------------------------------------
         // Etape 2 : Waiting for start cycle
         //----------------------------------------------
          IF TRUE                            AND
             ( stCycBundTilt.bTestOn         OR
               NOT(stCycBundTilt.bModTest) ) THEN
            stCycBundTilt.iStep := C_iSTEP_2 ;

            // Action Step 2
            stCycBundTilt.bTestOn := 0 ;

            //Waiting for start cycle
          END_IF

        C_iSTEP_2 :
         //----------------------------------------------
         // Etape 4 : Rising Tilter
         //----------------------------------------------
          IF g_bBund_StartTilt              AND
             g_bBundInitTilt_OK             AND
             ( stCycBundTilt.bTestOn        OR
              NOT(stCycBundTilt.bModTest) ) THEN
            stCycBundTilt.iStep := C_iSTEP_4 ;

            // Action Step 4
            stCycBundTilt.bTestOn := 0 ;

            bQ_Bund_DriveStart     := 1 ;
            bQ_Bund_DriveDirection := 1 ;
            g_bBund_StartTilt      := 0 ;
          END_IF

        C_iSTEP_4 :
         //----------------------------------------------
         // Step 5 : Move in cylinder 14C4 and 14C3
         //----------------------------------------------
          IF ( rPosTiltAct >= gr_rPosTilt14C4In ) AND
             ( stCycBundTilt.bTestOn              OR
               NOT(stCycBundTilt.bModTest) )      THEN
            stCycBundTilt.iStep := C_iSTEP_5 ;

            // Action Step 5
            stCycBundTilt.bTestOn := 0 ;

            bQ_Bund_SOL_14C3Out := 0; //;;;;;;;;;;;;modif 12092011 input also 14C3
            bQ_Bund_SOL_14C4Out := 0 ;
          END_IF

        C_iSTEP_5 :
         //----------------------------------------------
         // Step 6 : Output cylinder 14C4
         //          and waiting for Stop position
         //----------------------------------------------
          IF gI_Bund_S110                       AND
             ( rPosTiltAct >= rPosTilt14C4Out ) AND
             ( stCycBundTilt.bTestOn            OR
               NOT(stCycBundTilt.bModTest) )    THEN
            stCycBundTilt.iStep := C_iSTEP_6 ;

            // Action Step 6
            stCycBundTilt.bTestOn := 0 ;

            bQ_Bund_SOL_14C3Out  := 1;//;;;;;;;;;;;;modif 12092011
            bQ_Bund_SOL_14C4Out  := 1 ;
            g_bBund_MoveInSep_OK := NOT(bInitTiltCycl) ;
            // Waiting for Stop position
          END_IF

        C_iSTEP_6 :
         //----------------------------------------------
         // Etape 7 : Stop Tilter and waiting stop
         //----------------------------------------------
          IF NOT(gI_Bund_S110)               AND
             ( bIndPosUpStop                 OR
               g_bBund_EndTravUp )           AND
             ( stCycBundTilt.bTestOn         OR
               NOT(stCycBundTilt.bModTest) ) THEN
            stCycBundTilt.iStep := C_iSTEP_7 ;

            // Action Step 7
            stCycBundTilt.bTestOn := 0 ;

            bQ_Bund_DriveStart := 0 ;
            // Waiting stop
          END_IF

        C_iSTEP_7 :
         //----------------------------------------------
         // Etape 8 : Move down Tilter
         //----------------------------------------------
          IF stTON_StopTilt.Q                AND
             ( stCycBundTilt.bTestOn         OR
               NOT(stCycBundTilt.bModTest) ) THEN
            stCycBundTilt.iStep := C_iSTEP_8 ;

            // Action Step 8
            stCycBundTilt.bTestOn := 0 ;

            bQ_Bund_DriveStart     := 1 ;
            bQ_Bund_DriveDirection := 0 ;
          END_IF

        C_iSTEP_8 :
         //----------------------------------------------
         // Etape 9 : Move in cylinder 14C3 and 14C4
         //           Out cylinder 14C5
         //----------------------------------------------
          IF ( rPosTiltAct <= 59.0 )             AND
             ( stCycBundTilt.bTestOn             OR
               NOT(stCycBundTilt.bModTest) )     THEN
            stCycBundTilt.iStep := C_iSTEP_9 ;

            // Action Step 9
            stCycBundTilt.bTestOn := 0 ;

            bQ_Bund_SOL_14C3Out := 0 ;
            //bQ_Bund_SOL_14C4Out := 0 ;
            bQ_Bund_SOL_14C5Out := 1 ;
          END_IF

        C_iSTEP_9 :
         //----------------------------------------------
         // Etape 10 : Waiting for Stop position down
         //----------------------------------------------
          IF gI_Bund_S104                    AND
             //gI_Bund_S110                    AND
             ( stCycBundTilt.bTestOn         OR
               NOT(stCycBundTilt.bModTest) ) THEN
            stCycBundTilt.iStep := C_iSTEP_10 ;

            // Action Step 10
            stCycBundTilt.bTestOn := 0 ;

            //Waiting for Stop position down
          END_IF

        C_iSTEP_10 :
         //----------------------------------------------
         // Etape 11 : Stop Tilter and waiting stop
         //----------------------------------------------
          IF bIndPosDownStop                 AND
             ( stCycBundTilt.bTestOn         OR
               NOT(stCycBundTilt.bModTest) ) THEN
            stCycBundTilt.iStep := C_iSTEP_11 ;

            // Action Step 11
            stCycBundTilt.bTestOn := 0 ;

            bQ_Bund_DriveStart := 0 ;
            // Waiting stop
          END_IF

        C_iSTEP_11 :
         //----------------------------------------------
         // Etape 12 : Move out cylinder 14C3 and 14C4
         //----------------------------------------------
          IF stTON_StopTilt.Q                AND
             ( stCycBundTilt.bTestOn         OR
               NOT(stCycBundTilt.bModTest) ) THEN
            stCycBundTilt.iStep := C_iSTEP_12 ;

            // Action Step 12
            stCycBundTilt.bTestOn := 0 ;

            bQ_Bund_SOL_14C3Out := 1 ;
            bQ_Bund_SOL_14C4Out := 1 ;
          END_IF

        C_iSTEP_12 :
         //----------------------------------------------
         // Etape 13 : Waiting back of cylinder 14C5
         //----------------------------------------------
          IF NOT(gI_Bund_S104)               AND
             NOT(gI_Bund_S110)               AND
             ( stCycBundTilt.bTestOn         OR
               NOT(stCycBundTilt.bModTest) ) THEN
            stCycBundTilt.iStep := C_iSTEP_13 ;

            // Action Step 13
            stCycBundTilt.bTestOn := 0 ;

            // Waiting back of cylinder 14C5
          END_IF

        C_iSTEP_13 :
         //----------------------------------------------
         // Etape 2 : Waiting for start cycle
         //----------------------------------------------
         IF TRUE THEN
          //IF gI_Bund_S111                    AND   //MODIF DU 14092011  Cycle time too long
          //   ( stCycBundTilt.bTestOn         OR
          //     NOT(stCycBundTilt.bModTest) ) THEN
            stCycBundTilt.iStep := C_iSTEP_2 ;

            // Action Step 2
            stCycBundTilt.bTestOn := 0 ;
            //Waiting for start cycle

            g_bBund_InitTilt   := 0 ;
            bInitTiltCycl      := 0 ;
            g_bBundInitTilt_OK := 1 ;
          END_IF

        C_iSTEP_15 :
         //----------------------------------------------
         // Etape 16 : Rising Tilter
         //----------------------------------------------
          IF NOT(gI_Bund_S104)               AND
             NOT(gI_Bund_S110)               AND
             stTON_Out14C3.Q                 AND
             ( stCycBundTilt.bTestOn         OR
               NOT(stCycBundTilt.bModTest) ) THEN
            stCycBundTilt.iStep := C_iSTEP_16 ;
            // Action Step 4
            stCycBundTilt.bTestOn := 0 ;

            bQ_Bund_DriveStart     := 1 ;
            bQ_Bund_DriveDirection := 1 ;
            g_bBundInitTilt_OK     := 0 ;
            g_bBund_StartTilt      := 0 ;
          END_IF

        C_iSTEP_16 :
         //----------------------------------------------
         // Etape 7 : Stop Tilter and waiting stop
         //----------------------------------------------
          IF ( bIndPosUpStop                 OR
               g_bBund_EndTravUp )           AND
             ( stCycBundTilt.bTestOn         OR
               NOT(stCycBundTilt.bModTest) ) THEN
            stCycBundTilt.iStep := C_iSTEP_7 ;

            // Action Step 7
            stCycBundTilt.bTestOn := 0 ;

            bQ_Bund_DriveStart := 0 ;
            // Waiting stop
          END_IF

        C_iSTEP_25 :
         //----------------------------------------------
         // Etape 1 : Initialisation cycle
         //----------------------------------------------
          IF NOT(g_bIndBundManu)             AND
             ( stCycBundTilt.bTestOn         OR
               NOT(stCycBundTilt.bModTest) ) THEN
            stCycBundTilt.iStep := C_iSTEP_1 ;

            // Action Step 1
            stCycBundTilt.bTestOn := 0 ;

            stCycBundTilt.bFCyc := 0 ;
            stCycBundTilt.bCyc  := 1 ;
          END_IF
        END_CASE
    //---------------------------------------------------------------------------------------------------------------------

END_PROGRAM
```

### Program Logical/BagMachine_Section/BagBundler/Test_Simul (IEC) - A new program

#### Test_Simul.var
```iecst
(********************************************************************
 * COPYRIGHT -- .
 ********************************************************************
 * Program: Test_Simul
 * File: Test_Simul.var
 * Author: dominique
 * Created: August 20, 2011
 ********************************************************************
 * Local variables of program Test_Simul
 ********************************************************************)

VAR

  HGW_3StateIND1_0 : HGW_3StateIND1 ;
  bTest_ : ARRAY[0..9] OF BOOL ;
  H_FB_WS_S104 : H_FB_WatchSensor ;
  H_FB_Flash_0 : H_FB_Flash ;
END_VAR

VAR RETAIN
  iTest_ : ARRAY[0..9] OF INT ;
END_VAR

VAR CONSTANT

END_VAR
```

#### Test_SimulCyclic.st
```iecst
(********************************************************************
 * COPYRIGHT -- .
 ********************************************************************
 * Program: Test_Simul
 * File: Test_SimulCyclic.st
 * Author: dominique
 * Created: August 20, 2011
 ********************************************************************
 * Implementation of program Test_Simul
 ********************************************************************)

PROGRAM _CYCLIC

END_PROGRAM
```

#### Test_SimulInit.st
```iecst
(********************************************************************
 * COPYRIGHT -- .
 ********************************************************************
 * Program: Test_Simul
 * File: Test_SimulInit.st
 * Author: dominique
 * Created: August 20, 2011
 ********************************************************************
 * Implementation of program Test_Simul
 ********************************************************************)

PROGRAM _INIT

(* TODO : Add your code here *)

END_PROGRAM
```

### Program Logical/BagMachine_Section/ColdGlue (IEC)

#### ColdGlueCyclic.st - Cyclic code
```iecst
(********************************************************************
 * COPYRIGHT -- Microsoft
 ********************************************************************
 * Program: ColdGlue
 * File: ColdGlueCyclic.st
 * Author: pkiel
 * Created: July 13, 2011
 ********************************************************************
 * Implementation of program ColdGlue
 ********************************************************************)

PROGRAM _CYCLIC

(* Glue Off/On From HMI *)
	HGW_2StatePB_0.PB := EDGEPOS(Glue_PB);
	GlueText_Ind := HGW_2StatePB_0.Text_Ind;
	GlueColor_Ind := HGW_2StatePB_0.Color_Ind;
	Glue_On := HGW_2StatePB_0.State1;
	HGW_2StatePB_0();

(* Glue Manual/Auto From HMI *)
	HGW_2StatePB_1.PB := (EDGEPOS(GlueAuto_PB) OR (NOT Glue_Auto AND gA[9].Ind_InMotion));
	GlueAutoText_Ind := HGW_2StatePB_1.Text_Ind;
	GlueAutoColor_Ind := HGW_2StatePB_1.Color_Ind;
	Glue_Auto := HGW_2StatePB_1.State1;
	HGW_2StatePB_1();

(* Glue Auto Pressure Based On Machine Speed *)
	HGW_ScaleReal_0.Enable := Glue_Auto;
	HGW_ScaleReal_0.InputMin := 0.0;
	HGW_ScaleReal_0.InputMax := 1000.0;
	HGW_ScaleReal_0.InputRaw := gActualMachineSpeed_FPM;
	HGW_ScaleReal_0.ScaledMin := LIMIT (0,gSP_ColdGlue.MinPressure,400);
	HGW_ScaleReal_0.ScaledMax := LIMIT (0,gSP_ColdGlue.MaxPressure,400);
	PressureCmd := HGW_ScaleReal_0.ScaledOut;
	HGW_ScaleReal_0();

(* Glue Manual Pressure *)
	IF (NOT Glue_Auto) THEN
		PressureCmd := gSP_ColdGlue.ManPressure;
	END_IF

(* Glue Pressure Command Limit 0-100% *)
	PressureCmd := LIMIT (0,PressureCmd, 100);

(* If Disabled, Reduce Pressure To Zero  *)
	IF (NOT Glue_On) THEN
		PressureCmd := 0;
	END_IF

(* Generate Analog Command To Seam Paste System Pressure *)
	HGW_ScaleReal_1.Enable := 1;
	HGW_ScaleReal_1.InputMin := 0.0;
	HGW_ScaleReal_1.InputMax := 100.0;
	HGW_ScaleReal_1.InputRaw := PressureCmd;
	HGW_ScaleReal_1.ScaledMin := 0.0;
	HGW_ScaleReal_1.ScaledMax := 32767.0;
	//gQ_CMD_ColdGluePressure := REAL_TO_INT(HGW_ScaleReal_1.ScaledOut);
  gQ_CMD_RS_GluePressure  := REAL_TO_INT(HGW_ScaleReal_1.ScaledOut);
	HGW_ScaleReal_1();

(* Glue Auto On *)
  IF ((gActualMachineSpeed_FPM>=gSP_ColdGlue.AutoOnSpeed) AND gA[9].Ind_InMotion AND Glue_On AND gBagMachine_WebBreakOK) THEN
		GlueAuto_On := 1;
	ELSE
		GlueAuto_On := 0;
	END_IF

(* Glue Gun Clean Control *)
	HGW_Toggle_0(In := GlueClean_PB , Time := T#12ms);

(* Glue Gun Control *)
	IF ((GlueAuto_On OR GluePurge_PB OR HGW_Toggle_0.Out) AND gAlarmsOK AND gI_SS_SeamGlueOnOff) THEN
		gQ_CR_ColdGlue := 1;
	ELSE
		gQ_CR_ColdGlue := 0;
	END_IF

(* Is 2nd Tube Selected *)
	IF (gSP_TubeSelect) THEN
		gQ_CR_ColdGlueSelect := 1;
	ELSE
		gQ_CR_ColdGlueSelect := 0;
	END_IF

END_PROGRAM
```

#### ColdGlueInit.st - Initialization code
```iecst
(********************************************************************
 * COPYRIGHT -- Microsoft
 ********************************************************************
 * Program: ColdGlue
 * File: ColdGlueInit.st
 * Author: pkiel
 * Created: July 13, 2011
 ********************************************************************
 * Implementation of program ColdGlue
 ********************************************************************)

PROGRAM _INIT

(* Glue Off/On PB Colors *)
	HGW_2StatePB_0.BackColor_State0 := gBlue;
	HGW_2StatePB_0.ForeColor_State0 := gWhite;
	HGW_2StatePB_0.BackColor_State1 := gGreen;
	HGW_2StatePB_0.ForeColor_State1 := gBlack;

(* Glue Manual/Auto PB Colors *)
	HGW_2StatePB_1.BackColor_State0 := gYellow;
	HGW_2StatePB_1.ForeColor_State0 := gBlack;
	HGW_2StatePB_1.BackColor_State1 := gGreen;
	HGW_2StatePB_1.ForeColor_State1 := gBlack;

END_PROGRAM
```

#### ColdGlue.var - Local variables
```iecst
(********************************************************************
 * COPYRIGHT -- Microsoft
 ********************************************************************
 * Program: ColdGlue
 * File: ColdGlue.var
 * Author: pkiel
 * Created: July 13, 2011
 ********************************************************************
 * Local variables of program ColdGlue
 ********************************************************************)
VAR
	Glue_Auto : BOOL;
	Glue_On : BOOL;
	Glue_PB : BOOL;
	GlueAuto_On : BOOL;
	GlueAuto_PB : BOOL;
	GlueAutoColor_Ind : UINT;
	GlueAutoText_Ind : UINT;
	GlueColor_Ind : UINT;
	GluePurge_PB : BOOL;
	GlueText_Ind : UINT;
END_VAR
VAR RETAIN
	HGW_2StatePB_0 : HGW_2StatePB;
	HGW_2StatePB_1 : HGW_2StatePB;
END_VAR
VAR
	HGW_ScaleReal_0 : HGW_ScaleReal;
	HGW_ScaleReal_1 : HGW_ScaleReal;
	PressureCmd : REAL;
	GlueClean_PB : BOOL;
	HGW_Toggle_0 : HGW_Toggle;
END_VAR
```

### A8_Automat.var
```iecst
(********************************************************************
 * COPYRIGHT -- Microsoft
 ********************************************************************
 * Program: A8_Automat
 * File: A8_Automat.var
 * Author: dominique
 * Created: November 03, 2011
 ********************************************************************
 * Local variables of program A8_Automat
 ********************************************************************)
VAR
	AutData : MC_AUTDATA_TYP;
	AutomatStart : BOOL;
	ErrorID : UINT;
	MasterParID : UINT;
	MC_BR_AutControl_0 : MC_BR_AutControl;
	MC_BR_InitAutState_0 : MC_BR_InitAutState;
	MC_BR_InitMasterParIDTransfer_0 : MC_BR_InitMasterParIDTransfer;
	ParID_Ready : BOOL;
	Synch_Request : BOOL;
END_VAR
```

### Program Logical/BagMachine_Section/ColdMicroPerf/Axis8/A8_Basic (IEC)

#### A8_BasicInit.st - Initialization code
```iecst
(********************************************************************
 * COPYRIGHT -- Microsoft
 ********************************************************************
 * Program: A8_Basic
 * File: A8_BasicInit.st
 * Author: dominique
 * Created: November 03, 2011
 ********************************************************************
 * Implementation of program A8_Basic
 ********************************************************************)

PROGRAM _INIT

  g_iCMPerfType := C_i10DP ; // D.M. 07/11/2011     Brown_Paper_14606  Cold Micro Perf in 10Dp
  // Drive roll size calculation
  CASE g_iCMPerfType OF
    C_iM : ; // Case Metric
      g_rSizeCMPerfRol_mm := g_rZGearCMPerf_M * 10.0 ;
    C_i8DP : ; // Case 8DP
      g_rSizeCMPerfRol_mm := TRUNC(g_rZGearCMPerf_8DP*PI/8.0*25.4*1000.0)/1000.0 ;
    C_i10DP : ; // Case 10DP
      g_rSizeCMPerfRol_mm := TRUNC(g_rZGearCMPerf_10DP*PI/10.0*25.4*1000.0)/1000.0 ;
    C_i1_4P : ; // Case 1/4"
      g_rSizeCMPerfRol_mm := TRUNC(g_rZGearCMPerf_1_4P/4.0*25.4) ;
  END_CASE

	(* Axis Setpoint Variables *)
		gA[8].SP_MotorPPR := 12000;
		gA[8].SP_GearBoxInput:= 3;
		gA[8].SP_GearBoxOutput:= 1;
		gA[8].AxisPeriod := (gA[8].SP_MotorPPR*gA[8].SP_GearBoxInput/gA[8].SP_GearBoxOutput);
		gA[8].UnitsPerDeg := gA[8].AxisPeriod/360;
		gA[8].SP_Accel := 0.2*gA[8].AxisPeriod;
		gA[8].SP_Decel := 0.4*gA[8].AxisPeriod;
		gA[8].SP_EStopDecel := 1000.0*gA[8].AxisPeriod; // Stop axis from 1000 tr/min in 1s
		(* Theoretical Perimeter = 320mm *)
		gA[8].UnitsPerInch := (gA[8].AxisPeriod*25.4) / g_rSizeCMPerfRol_mm ;
    gA[8].rSP_CorPosVel := 0.0 ;
    gA[8].rSP_OverrideV := 1.0 ;
    gA[8].rSP_OverrideA := 1.0 ;
    gA[8].Cmd_EStopDisable := 0 ;

	(* access master axis *)
		AxisErrorNcAccess := ncaccess(ncACP10MAN, ADR('Axis8'), ADR(gA[8].Ident));

	(* Trigger Initialization Of ModPosition *)
		InitModPosition:=1;

END_PROGRAM
```

#### A8_Basic.var - Local variables
```iecst
(********************************************************************
 * COPYRIGHT -- Microsoft
 ********************************************************************
 * Program: A8_Basic
 * File: A8_Basic.var
 * Author: dominique
 * Created: November 03, 2011
 ********************************************************************
 * Local variables of program A8_Basic
 ********************************************************************)
VAR
	AutoAck : BOOL;
	AxisErrorNcAccess : UINT;
	DriveStatus : MC_DRIVESTATUS_TYP;
	HomeRestore : BOOL;
	InitEndlessPosition : BOOL;
	InitModPos_Done : BOOL;
	InitModPosition : BOOL;
	MC_BR_InitEndlessPosition_0 : MC_BR_InitEndlessPosition;
	MC_BR_InitModPos_0 : MC_BR_InitModPos;
	MC_BR_Phasing_0 : MC_BR_Phasing;
	MC_BR_ReadDriveStatus_0 : MC_BR_ReadDriveStatus;
	MC_Home_0 : MC_Home;
	MC_Home_1 : MC_Home;
	MC_MoveVelocity_0 : MC_MoveVelocity;
	MC_Power_0 : MC_Power;
	MC_ReadActualPosition_0 : MC_ReadActualPosition;
	MC_ReadActualTorque_0 : MC_ReadActualTorque;
	MC_ReadActualVelocity_0 : MC_ReadActualVelocity;
	MC_ReadAxisError_0 : MC_ReadAxisError;
	MC_ReadStatus_0 : MC_ReadStatus;
	MC_Reset_0 : MC_Reset;
	MC_Stop_0 : MC_Stop;
  MC_Stop_1 : MC_Stop;
  stTON_O : TON ;
	ResetError : BOOL;
  MC_SetOverride_0 : MC_SetOverride;
END_VAR
```

### A8_Control.var
```iecst
(********************************************************************
 * COPYRIGHT -- Microsoft
 ********************************************************************
 * Program: A8_Control
 * File: A8_Control.var
 * Author: dominique
 * Created: November 03, 2011
 ********************************************************************
 * Local variables of program A8_Control
 ********************************************************************)
VAR
	Synch_Permissive : BOOL;
	TOF_0 : TOF;
END_VAR
```

### Program Logical/BagMachine_Section/ColdMicroPerf/Axis8/A8_Draw

#### A8_DrawCyclic.st
```iecst
(********************************************************************
 * COPYRIGHT -- Microsoft
 ********************************************************************
 * Program: A8_Draw
 * File: A8_DrawCyclic.st
 * Author: dominique
 * Created: November 03, 2011
 ********************************************************************
 * Implementation of program A8_Draw
 ********************************************************************)

PROGRAM _CYCLIC

  // Draw Setpoint Limits
	gRecipeActive.rCMPerf_Draw := LIMIT(-100,gRecipeActive.rCMPerf_Draw,100);

(* Manual Draw Calculations *)
  IF ( ( (gRecipeActive.rCMPerf_Draw <> Draw_Old) OR
         (g_rSizeCMPerfRol_mm <> rSizeTool_Old)   OR
         (NOT First) )                            AND
         gA[8].Ind_SynchronizedMotion )           THEN
		gA8_GearValue := gA[8].AxisPeriod * g_rSizeEntryPullRol_mm/g_rSizeCMPerfRol_mm * (1.0+(gr_rMaxRangeWebDraw * 0.01 * gRecipeActive.rCMPerf_Draw * 0.01));
		Draw_Old := gRecipeActive.rCMPerf_Draw;
    rSizeTool_Old := g_rSizeCMPerfRol_mm ;
		First :=1;
		IF(gA[8].Ind_SynchronizedMotion) THEN
			gA[8].Cmd_SynchronizedMotionUpdate := 1;
		END_IF
	END_IF

END_PROGRAM
```

- Data object Logical/BagMachine_Section/ColdMicroPerf/Axis8/A8_Init (Ax) (no source held here)

- Data object Logical/BagMachine_Section/ColdMicroPerf/Axis8/A8_Par (Apt) (no source held here)

### Program Logical/BagMachine_Section/ColdMicroPerf/CMPerf_Gen (IEC)

#### CMPerf_GenCyclic.st - Cyclic code
```iecst
(********************************************************************
 * COPYRIGHT -- .
 ********************************************************************
 * Program: CMPerf_Gen
 * File: CMPerf_GenCyclic.st
 * Author: dominique
 * Created: November 05, 2011
 ********************************************************************
 * Implementation of program CMPerf_Gen
 ********************************************************************)

PROGRAM _CYCLIC

  // ----------------------------------------------------------------------------------
  // On/Off Cold Micro Perf
  // Cas On
  bOnReq := HMI_CMPerf_bOnOffPB AND NOT(gRecipeActive.bSelColdMicroPerfProd) ;
  IF bOnReq THEN
    IF NOT(gA[9].Ind_InMotion) AND
       1                       THEN
      gRecipeActive.bSelColdMicroPerfProd := 1 ;
    ELSE
      gRecipeActive.bSelColdMicroPerfProd := 0 ;
      HMI_CMPerf_bOnOffPB := 0 ;
    END_IF ;
  END_IF ;

  // Cas Off
  bOffReq := NOT(HMI_CMPerf_bOnOffPB) AND gRecipeActive.bSelColdMicroPerfProd ;
  IF bOffReq THEN
    IF NOT(gA[9].Ind_InMotion) AND
       1                       THEN
      gRecipeActive.bSelColdMicroPerfProd := 0 ;
    ELSE
      gRecipeActive.bSelColdMicroPerfProd := 1 ;
      HMI_CMPerf_bOnOffPB := 1 ;
    END_IF ;
  END_IF ;

  // ----------------------------------------------------------------------------------
  // Axis ativation
  gA[8].bActive := gRecipeActive.bSelColdMicroPerfProd ;

  // ----------------------------------------------------------------------------------
  // Tool size change lock
  bToolSizeLock := NOT(gA[9].Ind_InMotion)                  OR
                   NOT(gRecipeActive.bSelColdMicroPerfProd) ;

END_PROGRAM
```

- Program Logical/BagMachine_Section/Count (IEC) (no source held here)

### Data object Logical/BagMachine_Section/Drum/Axis7/A7_Init (Ax) - Servo Axis Initialization File

#### A7_Init.ax
```
InitParameter (Version=2.24.0, NcSwId=ACP10)
  ACP10AXIS_typ:
    dig_in:
      level:
        reference = ncACTIV_HI
        pos_hw_end = ncACTIV_HI
        neg_hw_end = ncACTIV_HI
        trigger1 = ncACTIV_HI
        trigger2 = ncACTIV_HI
    encoder_if:
      parameter:
        count_dir = ncSTANDARD
        scaling:
          load:
            units = 12000  // Units at the load = 36000 x 4 / 12          x 4 because 4 bags for 1 revolution of the Drum, Drum Axis performs 4 x 36000 units per revolution
            rev_motor = 1  // Motor revolutions = 1
    limit:
      parameter:
        v_pos = 600000.0
        v_neg = 600000.0
        a1_pos = 5e+006
        a2_pos = 5e+006
        a1_neg = 5e+006
        a2_neg = 5e+006
        t_jolt = 0.0
        t_in_pos = 0.5
        pos_sw_end = 8388607
        neg_sw_end = -8388608
        ds_warning = 500.0
        ds_stop = 1000.0
        a_stop = 1e+030
        dv_stop = 0
        dv_stop_mode = ncOFF
    controller:
      mode = ncPOSITION
      position:
        kv = 300.0
        tn = 0.0
        t_predict = 0.0004
        t_total = 0.0012
        p_max = 1e+030
        i_max = 0.0
      speed:
        kv = 30.0
        tn = 0.0
        t_filter = 0.0
        isq_filter1:
          type = ncOFF
          a0 = 0.0
          a1 = 0.0
          b0 = 0.0
          b1 = 0.0
          b2 = 0.0
          c0_par_id = 0
          c1_par_id = 0
        isq_filter2:
          type = ncOFF
          a0 = 0.0
          a1 = 0.0
          b0 = 0.0
          b1 = 0.0
          b2 = 0.0
          c0_par_id = 0
          c1_par_id = 0
        isq_filter3:
          type = ncOFF
          a0 = 0.0
          a1 = 0.0
          b0 = 0.0
          b1 = 0.0
          b2 = 0.0
          c0_par_id = 0
          c1_par_id = 0
      uf:
        type = ncLINEAR
        auto_config = ncMOTOR_PAR
        u0 = 0.0
        un = 0.0
        fn = 50.0
        k_f_slip = 0.0
      ff:
        torque_load = 0.0
        torque_pos = 0.0
        torque_neg = 0.0
        kv_torque = 0.0
        inertia = 0.0
        t_filter_a = 0.0
    move:
      stop:
        parameter[0]:
          decel_ramp = ncA_LIMIT
          controller = ncON
        parameter[1]:
          decel_ramp = ncA_LIMIT
          controller = ncON
        parameter[2]:
          decel_ramp = ncA_LIMIT
          controller = ncON
        parameter[3]:
          decel_ramp = ncA_LIMIT
          controller = ncON
        quickstop:
          decel_ramp = ncA_LIMIT
        drive_error:
          decel_ramp = ncA_LIMIT
      homing:
        parameter:
          s = 0
          v_switch = 3600.0
          v_trigger = 360.0
          a = 50000.0
          mode = ncHOME_OFFSET
          edge_sw = ncPOSITIVE
          start_dir = ncPOSITIVE
          trigg_dir = ncPOSITIVE
          ref_pulse = ncOFF
          tr_s_block = 0.0
      basis:
        parameter:
          v_pos = 36000.0
          v_neg = 100000.0
          a1_pos = 50000.0
          a2_pos = 50000.0
          a1_neg = 50000.0
          a2_neg = 50000.0
    message:
      text:
        parameter:
          format = ncBREAK
          columns = 80
          data_modul = Error_Eng
```

### Program Logical/BagMachine_Section/Drum/Axis7/A7_Basic (IEC) - Basic Servo
